C07176=1030.906,187.234,-109.081,169.495,44.538,158.415
C07177=1030.900,186.985,-109.057,169.491,44.540,158.415
C07178=1030.894,186.736,-109.033,169.489,44.542,158.415
C07179=1030.888,186.488,-109.009,169.485,44.543,158.415
C07180=1030.882,186.238,-108.984,169.482,44.545,158.415
C07181=1030.877,185.990,-108.961,169.478,44.546,158.415
C07182=1030.870,185.741,-108.938,169.475,44.549,158.415
C07183=1030.865,185.492,-108.913,169.472,44.550,158.415
C07184=1030.859,185.244,-108.889,169.468,44.552,158.415
C07185=1030.854,184.995,-108.866,169.466,44.553,158.415
C07186=1030.847,184.746,-108.842,169.462,44.555,158.415
C07187=1030.842,184.497,-108.818,169.458,44.557,158.415
C07188=1030.836,184.249,-108.794,169.456,44.559,158.415
C07189=1030.829,183.999,-108.771,169.452,44.560,158.415
C07190=1030.824,183.751,-108.746,169.449,44.562,158.415
C07191=1030.818,183.502,-108.723,169.445,44.564,158.415
C07192=1030.813,183.253,-108.699,169.442,44.566,158.415
C07193=1030.806,183.004,-108.675,169.439,44.567,158.415
C07194=1030.800,182.756,-108.651,169.435,44.569,158.415
C07195=1030.795,182.507,-108.629,169.433,44.571,158.416
C07196=1030.788,182.257,-108.605,169.429,44.573,158.416
C07197=1030.781,182.009,-108.582,169.426,44.575,158.416
C07198=1030.776,181.760,-108.559,169.423,44.577,158.416
C07199=1030.769,181.511,-108.535,169.419,44.579,158.416
C07200=1030.763,181.263,-108.512,169.416,44.581,158.416
C07201=1030.758,181.014,-108.489,169.413,44.583,158.416
C07202=1030.751,180.765,-108.465,169.410,44.585,158.416
C07203=1030.744,180.516,-108.443,169.406,44.587,158.416
C07204=1030.739,180.267,-108.420,169.403,44.588,158.416
C07205=1030.732,180.018,-108.396,169.400,44.591,158.416
C07206=1030.726,179.769,-108.373,169.396,44.593,158.417
C07207=1030.720,179.521,-108.349,169.394,44.595,158.417
C07208=1030.714,179.271,-108.326,169.390,44.597,158.417
C07209=1030.708,179.023,-108.304,169.387,44.599,158.417
C07210=1030.702,178.774,-108.281,169.384,44.601,158.417
C07211=1030.696,178.526,-108.257,169.380,44.602,158.417
C07212=1030.689,178.276,-108.234,169.377,44.604,158.417
C07213=1030.684,178.027,-108.211,169.374,44.606,158.417
C07214=1030.677,177.779,-108.188,169.370,44.608,158.417
C07215=1030.671,177.530,-108.165,169.368,44.610,158.417
C07216=1030.665,177.281,-108.141,169.364,44.613,158.417
C07217=1030.659,177.032,-108.119,169.362,44.614,158.418
C07218=1030.653,176.783,-108.096,169.358,44.616,158.418
C07219=1030.647,176.535,-108.073,169.355,44.618,158.418
C07220=1030.640,176.285,-108.049,169.352,44.620,158.418
C07221=1030.635,176.036,-108.026,169.348,44.622,158.418
C07222=1030.629,175.788,-108.003,169.346,44.624,158.418
C07223=1030.623,175.539,-107.980,169.342,44.626,158.418
C07224=1030.616,175.291,-107.957,169.339,44.628,158.418
C07225=1030.610,175.041,-107.934,169.336,44.630,158.418
C07226=1030.604,174.792,-107.911,169.333,44.632,158.418
C07227=1030.599,174.543,-107.888,169.329,44.634,158.418
C07228=1030.593,174.294,-107.865,169.326,44.636,158.419
C07229=1030.586,174.046,-107.843,169.323,44.638,158.419
C07230=1030.581,173.797,-107.820,169.320,44.640,158.419
C07231=1030.574,173.548,-107.796,169.317,44.642,158.419
C07232=1030.568,173.299,-107.773,169.314,44.644,158.419
C07233=1030.563,173.050,-107.750,169.311,44.646,158.419
C07234=1030.556,172.766,-107.724,169.307,44.648,158.419
C07235=1030.549,172.483,-107.698,169.304,44.650,158.419
C07236=1030.542,172.199,-107.672,169.300,44.652,158.419
C07237=1030.535,171.914,-107.646,169.297,44.655,158.420
C07238=1030.529,171.665,-107.623,169.293,44.657,158.420
C07239=1030.524,171.417,-107.600,169.291,44.659,158.420
C07240=1030.517,171.168,-107.578,169.287,44.661,158.420
C07241=1030.511,170.919,-107.555,169.284,44.663,158.420
C07242=1030.506,170.670,-107.532,169.281,44.665,158.420
C07243=1030.499,170.421,-107.509,169.278,44.667,158.420
C07244=1030.494,170.172,-107.486,169.275,44.669,158.420
C07245=1030.487,169.923,-107.463,169.272,44.671,158.420
C07246=1030.481,169.674,-107.440,169.269,44.673,158.421
C07247=1030.476,169.425,-107.418,169.266,44.674,158.421
C07248=1030.470,169.176,-107.395,169.262,44.676,158.421
C07249=1030.463,168.928,-107.372,169.260,44.678,158.421
C07250=1030.458,168.679,-107.349,169.256,44.681,158.421
C07251=1030.452,168.430,-107.326,169.254,44.682,158.421
C07252=1030.446,168.181,-107.303,169.250,44.685,158.421
C07253=1030.440,167.933,-107.281,169.247,44.687,158.421
C07254=1030.434,167.683,-107.259,169.244,44.689,158.421
C07255=1030.429,167.434,-107.236,169.241,44.691,158.421
C07256=1030.423,167.185,-107.213,169.239,44.693,158.422
C07257=1030.416,166.937,-107.191,169.235,44.695,158.422
C07258=1030.411,166.688,-107.168,169.233,44.697,158.422
C07259=1030.405,166.439,-107.145,169.229,44.698,158.422
C07260=1030.399,166.190,-107.122,169.226,44.700,158.422
C07261=1030.393,165.941,-107.100,169.223,44.702,158.422
C07262=1030.387,165.692,-107.077,169.220,44.704,158.422
C07263=1030.382,165.443,-107.054,169.217,44.706,158.422
C07264=1030.376,165.194,-107.031,169.214,44.708,158.422
C07265=1030.369,164.945,-107.009,169.211,44.710,158.423
C07266=1030.364,164.696,-106.987,169.208,44.712,158.423
C07267=1030.358,164.447,-106.964,169.205,44.714,158.423
C07268=1030.353,164.199,-106.941,169.202,44.716,158.423
C07269=1030.347,163.950,-106.919,169.199,44.718,158.423
C07270=1030.341,163.701,-106.896,169.197,44.720,158.423
C07271=1030.335,163.452,-106.874,169.193,44.722,158.423
C07272=1030.330,163.203,-106.851,169.190,44.724,158.423
C07273=1030.323,162.954,-106.828,169.188,44.726,158.423
C07274=1030.318,162.705,-106.806,169.184,44.728,158.423
C07275=1030.312,162.456,-106.783,169.181,44.730,158.424
C07276=1030.306,162.207,-106.761,169.178,44.732,158.424
C07277=1030.300,161.958,-106.738,169.175,44.734,158.424
C07278=1030.295,161.710,-106.716,169.173,44.736,158.424
C07279=1030.289,161.461,-106.693,169.169,44.738,158.424
C07280=1030.283,161.212,-106.671,169.167,44.740,158.424
C07281=1030.277,160.963,-106.648,169.164,44.742,158.424
C07282=1030.272,160.714,-106.626,169.160,44.744,158.424
C07283=1030.266,160.465,-106.604,169.158,44.746,158.425
C07284=1030.260,160.216,-106.581,169.155,44.748,158.425
C07285=1030.255,159.967,-106.558,169.152,44.749,158.425
C07286=1030.249,159.718,-106.536,169.149,44.751,158.425
C07287=1030.243,159.469,-106.514,169.145,44.754,158.425
C07288=1030.237,159.220,-106.492,169.143,44.756,158.425
C07289=1030.231,158.971,-106.469,169.141,44.758,158.425
C07290=1030.225,158.722,-106.448,169.137,44.760,158.425
C07291=1030.218,158.473,-106.425,169.134,44.762,158.425
C07292=1030.213,158.224,-106.403,169.131,44.764,158.426
C07293=1030.207,157.975,-106.382,169.128,44.766,158.426
C07294=1030.201,157.727,-106.359,169.126,44.769,158.426
C07295=1030.195,157.477,-106.337,169.122,44.771,158.426
C07296=1030.189,157.229,-106.315,169.120,44.773,158.426
C07297=1030.183,156.980,-106.293,169.116,44.775,158.426
C07298=1030.176,156.695,-106.267,169.113,44.777,158.426
C07299=1030.170,156.411,-106.243,169.110,44.780,158.427
C07300=1030.162,156.127,-106.218,169.107,44.782,158.427
C07301=1030.156,155.842,-106.193,169.103,44.785,158.427
C07302=1030.149,155.593,-106.170,169.100,44.787,158.427
C07303=1030.144,155.344,-106.149,169.097,44.789,158.427
C07304=1030.138,155.095,-106.127,169.095,44.791,158.427
C07305=1030.132,154.846,-106.105,169.091,44.794,158.428
C07306=1030.126,154.597,-106.083,169.089,44.796,158.428
C07307=1030.120,154.348,-106.061,169.086,44.798,158.428
C07308=1030.115,154.099,-106.039,169.083,44.800,158.428
C07309=1030.108,153.851,-106.017,169.080,44.802,158.428
C07310=1030.102,153.601,-105.995,169.078,44.804,158.428
C07311=1030.096,153.352,-105.974,169.074,44.807,158.429
C07312=1030.091,153.103,-105.952,169.072,44.808,158.429
C07313=1030.085,152.855,-105.930,169.068,44.811,158.429
C07314=1030.078,152.606,-105.908,169.066,44.813,158.429
C07315=1030.072,152.356,-105.886,169.063,44.815,158.429
C07316=1030.066,152.107,-105.865,169.060,44.817,158.429
C07317=1030.060,151.859,-105.843,169.057,44.819,158.429
C07318=1030.054,151.609,-105.822,169.055,44.821,158.430
C07319=1030.049,151.360,-105.799,169.051,44.823,158.430
C07320=1030.042,151.111,-105.777,169.049,44.826,158.430
C07321=1030.037,150.863,-105.756,169.046,44.828,158.430
C07322=1030.031,150.614,-105.734,169.043,44.830,158.430
C07323=1030.025,150.364,-105.713,169.040,44.832,158.430
C07324=1030.018,150.115,-105.691,169.038,44.835,158.431
C07325=1030.013,149.867,-105.670,169.034,44.837,158.431
C07326=1030.007,149.617,-105.648,169.032,44.839,158.431
C07327=1030.000,149.368,-105.627,169.029,44.841,158.431
C07328=1029.996,149.119,-105.605,169.026,44.844,158.431
C07329=1029.989,148.870,-105.583,169.023,44.846,158.431
C07330=1029.983,148.621,-105.561,169.021,44.848,158.431
C07331=1029.977,148.373,-105.539,169.017,44.850,158.431
C07332=1029.971,148.124,-105.518,169.015,44.852,158.432
C07333=1029.965,147.875,-105.496,169.012,44.854,158.432
C07334=1029.959,147.626,-105.475,169.009,44.856,158.432
C07335=1029.953,147.377,-105.453,169.006,44.858,158.432
C07336=1029.948,147.127,-105.432,169.004,44.861,158.432
C07337=1029.941,146.878,-105.411,169.000,44.863,158.433
C07338=1029.936,146.629,-105.389,168.998,44.865,158.433
C07339=1029.930,146.380,-105.368,168.995,44.867,158.433
C07340=1029.924,146.131,-105.346,168.992,44.870,158.433
C07341=1029.918,145.883,-105.325,168.989,44.872,158.433
C07342=1029.912,145.633,-105.303,168.987,44.874,158.433
C07343=1029.905,145.384,-105.282,168.983,44.877,158.434
C07344=1029.899,145.136,-105.261,168.981,44.879,158.434
C07345=1029.893,144.887,-105.239,168.978,44.881,158.434
C07346=1029.887,144.637,-105.218,168.975,44.883,158.434
C07347=1029.882,144.388,-105.197,168.972,44.885,158.434
C07348=1029.876,144.139,-105.175,168.970,44.888,158.434
C07349=1029.869,143.890,-105.154,168.967,44.890,158.435
C07350=1029.863,143.642,-105.133,168.964,44.892,158.435
C07351=1029.857,143.392,-105.112,168.962,44.895,158.435
C07352=1029.852,143.143,-105.091,168.959,44.897,158.435
C07353=1029.846,142.894,-105.069,168.955,44.899,158.435
C07354=1029.839,142.645,-105.048,168.953,44.901,158.435
C07355=1029.834,142.397,-105.026,168.951,44.903,158.436
C07356=1029.828,142.147,-105.006,168.947,44.906,158.436
C07357=1029.822,141.899,-104.985,168.945,44.908,158.436
C07358=1029.815,141.649,-104.963,168.942,44.910,158.436
C07359=1029.809,141.400,-104.942,168.940,44.912,158.436
C07360=1029.804,141.151,-104.921,168.936,44.915,158.436
C07361=1029.798,140.902,-104.899,168.934,44.917,158.437
C07362=1029.791,140.618,-104.875,168.930,44.920,158.437
C07363=1029.784,140.333,-104.851,168.928,44.922,158.437
C07364=1029.778,140.047,-104.827,168.924,44.925,158.437
C07365=1029.771,139.763,-104.803,168.921,44.927,158.437
C07366=1029.765,139.514,-104.781,168.919,44.929,158.438
C07367=1029.759,139.265,-104.761,168.916,44.931,158.438
C07368=1029.753,139.016,-104.740,168.913,44.934,158.438
C07369=1029.747,138.768,-104.718,168.910,44.936,158.438
C07370=1029.741,138.518,-104.697,168.908,44.938,158.438
C07371=1029.735,138.269,-104.677,168.905,44.941,158.438
C07372=1029.729,138.020,-104.656,168.902,44.943,158.439
C07373=1029.723,137.770,-104.634,168.899,44.946,158.439
C07374=1029.717,137.522,-104.613,168.897,44.947,158.439
C07375=1029.711,137.272,-104.593,168.893,44.950,158.439
C07376=1029.705,137.024,-104.571,168.891,44.952,158.439
C07377=1029.699,136.774,-104.551,168.888,44.954,158.439
C07378=1029.693,136.526,-104.530,168.886,44.957,158.440
C07379=1029.687,136.276,-104.509,168.883,44.959,158.440
C07380=1029.681,136.028,-104.488,168.880,44.962,158.440
C07381=1029.675,135.778,-104.467,168.878,44.964,158.440
C07382=1029.669,135.530,-104.446,168.875,44.966,158.440
C07383=1029.663,135.280,-104.426,168.872,44.968,158.441
C07384=1029.657,135.032,-104.404,168.869,44.970,158.441
C07385=1029.651,134.782,-104.384,168.867,44.973,158.441
C07386=1029.645,134.534,-104.363,168.864,44.975,158.441
C07387=1029.638,134.284,-104.342,168.861,44.978,158.441
C07388=1029.633,134.035,-104.322,168.859,44.980,158.442
C07389=1029.627,133.786,-104.300,168.856,44.982,158.442
C07390=1029.621,133.537,-104.280,168.854,44.984,158.442
C07391=1029.615,133.288,-104.259,168.850,44.987,158.442
C07392=1029.609,133.039,-104.239,168.848,44.989,158.442
C07393=1029.603,132.789,-104.218,168.845,44.991,158.442
C07394=1029.597,132.541,-104.197,168.843,44.994,158.443
C07395=1029.591,132.292,-104.176,168.839,44.996,158.443
C07396=1029.585,132.043,-104.155,168.837,44.999,158.443
C07397=1029.579,131.794,-104.135,168.834,45.001,158.443
C07398=1029.573,131.544,-104.114,168.832,45.003,158.443
C07399=1029.567,131.296,-104.093,168.830,45.005,158.444
C07400=1029.561,131.046,-104.072,168.826,45.007,158.444
C07401=1029.555,130.797,-104.052,168.824,45.010,158.444
C07402=1029.550,130.549,-104.031,168.821,45.012,158.444
C07403=1029.543,130.299,-104.011,168.819,45.015,158.444
C07404=1029.538,130.050,-103.990,168.815,45.017,158.445
C07405=1029.531,129.800,-103.970,168.813,45.019,158.445
C07406=1029.525,129.552,-103.950,168.810,45.021,158.445
C07407=1029.518,129.303,-103.929,168.808,45.024,158.445
C07408=1029.513,129.054,-103.908,168.805,45.027,158.445
C07409=1029.507,128.804,-103.888,168.802,45.029,158.446
C07410=1029.501,128.555,-103.868,168.800,45.032,158.446
C07411=1029.494,128.306,-103.848,168.797,45.033,158.446
C07412=1029.488,128.057,-103.828,168.794,45.036,158.446
C07413=1029.482,127.808,-103.807,168.792,45.038,158.446
C07414=1029.476,127.559,-103.786,168.789,45.041,158.447
C07415=1029.470,127.310,-103.766,168.787,45.044,158.447
C07416=1029.463,127.061,-103.746,168.783,45.046,158.447
C07417=1029.458,126.811,-103.725,168.781,45.048,158.447
C07418=1029.452,126.563,-103.705,168.779,45.050,158.447
C07419=1029.445,126.313,-103.685,168.776,45.053,158.448
C07420=1029.439,126.064,-103.665,168.773,45.056,158.448
C07421=1029.434,125.814,-103.644,168.770,45.058,158.448
C07422=1029.427,125.566,-103.624,168.768,45.060,158.448
C07423=1029.421,125.317,-103.604,168.766,45.062,158.448
C07424=1029.415,125.068,-103.583,168.763,45.065,158.449
C07425=1029.409,124.819,-103.563,168.760,45.067,158.449
C07426=1029.403,124.575,-103.543,168.757,45.070,158.449
C07427=1029.397,124.332,-103.524,168.755,45.072,158.449
C07428=1029.391,124.088,-103.504,168.752,45.075,158.450
C07429=1029.386,123.845,-103.484,168.750,45.077,158.450
C07430=1029.380,123.602,-103.464,168.748,45.079,158.450
C07431=1029.374,123.358,-103.445,168.744,45.081,158.450
C07432=1029.368,123.115,-103.425,168.742,45.084,158.450
C07433=1029.362,122.871,-103.405,168.739,45.086,158.450
C07434=1029.356,122.622,-103.385,168.737,45.089,158.451
C07435=1029.350,122.373,-103.365,168.734,45.091,158.451
C07436=1029.344,122.124,-103.345,168.732,45.093,158.451
C07437=1029.337,121.875,-103.325,168.728,45.095,158.451
C07438=1029.332,121.625,-103.304,168.726,45.098,158.451
C07439=1029.326,121.377,-103.284,168.724,45.101,158.452
C07440=1029.320,121.127,-103.264,168.721,45.103,158.452
C07441=1029.314,120.878,-103.244,168.719,45.105,158.452
C07442=1029.308,120.629,-103.223,168.716,45.107,158.452
C07443=1029.302,120.380,-103.203,168.713,45.110,158.453
C07444=1029.296,120.131,-103.183,168.711,45.112,158.453
C07445=1029.290,119.882,-103.163,168.708,45.115,158.453
C07446=1029.284,119.633,-103.144,168.706,45.117,158.453
C07447=1029.279,119.383,-103.123,168.703,45.119,158.453
C07448=1029.272,119.134,-103.103,168.701,45.121,158.454
C07449=1029.266,118.885,-103.083,168.698,45.124,158.454
C07450=1029.260,118.636,-103.063,168.695,45.126,158.454
C07451=1029.254,118.388,-103.043,168.693,45.129,158.454
C07452=1029.248,118.138,-103.022,168.690,45.131,158.454
C07453=1029.242,117.889,-103.002,168.688,45.134,158.455
C07454=1029.235,117.592,-102.979,168.685,45.136,158.455
C07455=1029.229,117.296,-102.955,168.681,45.139,158.455
C07456=1029.221,117.001,-102.931,168.679,45.142,158.455
C07457=1029.214,116.704,-102.907,168.676,45.145,158.456
C07458=1029.208,116.455,-102.887,168.673,45.147,158.456
C07459=1029.202,116.206,-102.867,168.671,45.149,158.456
C07460=1029.197,115.957,-102.848,168.668,45.151,158.456
C07461=1029.190,115.707,-102.828,168.665,45.154,158.456
C07462=1029.185,115.458,-102.807,168.662,45.156,158.456
C07463=1029.179,115.209,-102.787,168.660,45.159,158.457
C07464=1029.173,114.960,-102.768,168.658,45.161,158.457
C07465=1029.167,114.711,-102.748,168.655,45.164,158.457
C07466=1029.161,114.462,-102.728,168.653,45.165,158.457
C07467=1029.155,114.213,-102.708,168.650,45.167,158.457
C07468=1029.150,113.963,-102.688,168.648,45.170,158.458
C07469=1029.144,113.714,-102.668,168.644,45.172,158.458
C07470=1029.138,113.465,-102.648,168.642,45.175,158.458
C07471=1029.132,113.217,-102.628,168.639,45.177,158.458
C07472=1029.126,112.967,-102.609,168.637,45.180,158.458
C07473=1029.119,112.718,-102.588,168.635,45.182,158.459
C07474=1029.114,112.468,-102.569,168.632,45.184,158.459
C07475=1029.108,112.219,-102.549,168.630,45.187,158.459
C07476=1029.102,111.971,-102.529,168.627,45.189,158.459
C07477=1029.096,111.721,-102.510,168.624,45.192,158.459
C07478=1029.090,111.472,-102.490,168.622,45.194,158.460
C07479=1029.084,111.222,-102.470,168.619,45.196,158.460
C07480=1029.078,110.973,-102.450,168.617,45.199,158.460
C07481=1029.072,110.724,-102.431,168.614,45.201,158.460
C07482=1029.065,110.475,-102.412,168.612,45.204,158.461
C07483=1029.059,110.227,-102.392,168.610,45.206,158.461
C07484=1029.054,109.977,-102.373,168.606,45.209,158.461
C07485=1029.048,109.728,-102.353,168.604,45.211,158.461
C07486=1029.041,109.478,-102.333,168.601,45.213,158.461
C07487=1029.035,109.229,-102.314,168.599,45.216,158.462
C07488=1029.029,108.980,-102.294,168.597,45.219,158.462
C07489=1029.023,108.731,-102.275,168.594,45.220,158.462
C07490=1029.016,108.447,-102.253,168.591,45.223,158.462
C07491=1029.009,108.162,-102.231,168.588,45.227,158.463
C07492=1029.002,107.877,-102.209,168.586,45.230,158.463
C07493=1028.995,107.591,-102.186,168.582,45.232,158.463
C07494=1028.989,107.342,-102.166,168.580,45.234,158.463
C07495=1028.983,107.093,-102.147,168.577,45.237,158.463
C07496=1028.977,106.844,-102.128,168.575,45.240,158.464
C07497=1028.971,106.595,-102.108,168.573,45.242,158.464
C07498=1028.965,106.345,-102.089,168.569,45.245,158.464
C07499=1028.959,106.096,-102.071,168.567,45.247,158.464
C07500=1028.953,105.847,-102.051,168.564,45.249,158.464
C07501=1028.947,105.598,-102.031,168.562,45.252,158.465
C07502=1028.941,105.349,-102.011,168.560,45.254,158.465
C07503=1028.935,105.100,-101.993,168.557,45.257,158.465
C07504=1028.929,104.851,-101.973,168.555,45.259,158.465
C07505=1028.922,104.601,-101.953,168.553,45.261,158.466
C07506=1028.916,104.352,-101.935,168.549,45.264,158.466
C07507=1028.910,104.102,-101.915,168.547,45.267,158.466
C07508=1028.905,103.853,-101.896,168.544,45.269,158.466
C07509=1028.899,103.604,-101.876,168.542,45.271,158.466
C07510=1028.892,103.355,-101.857,168.540,45.273,158.467
C07511=1028.886,103.106,-101.838,168.537,45.276,158.467
C07512=1028.880,102.857,-101.818,168.535,45.279,158.467
C07513=1028.874,102.608,-101.800,168.532,45.281,158.467
C07514=1028.868,102.358,-101.780,168.530,45.283,158.468
C07515=1028.863,102.109,-101.761,168.527,45.286,158.468
C07516=1028.857,101.860,-101.741,168.524,45.288,158.468
C07517=1028.850,101.611,-101.722,168.522,45.291,158.468
C07518=1028.845,101.362,-101.703,168.519,45.293,158.468
C07519=1028.839,101.112,-101.684,168.517,45.296,158.469
C07520=1028.832,100.864,-101.665,168.515,45.298,158.469
C07521=1028.826,100.614,-101.645,168.512,45.300,158.469
C07522=1028.821,100.365,-101.626,168.510,45.303,158.469
C07523=1028.815,100.115,-101.607,168.507,45.305,158.469
C07524=1028.809,99.866,-101.588,168.505,45.308,158.470
C07525=1028.803,99.617,-101.569,168.502,45.310,158.470
C07526=1028.796,99.368,-101.550,168.499,45.312,158.470
C07527=1028.791,99.119,-101.530,168.497,45.315,158.470
C07528=1028.784,98.870,-101.512,168.495,45.318,158.471
C07529=1028.778,98.621,-101.493,168.492,45.320,158.471
C07530=1028.772,98.371,-101.474,168.490,45.322,158.471
C07531=1028.766,98.122,-101.455,168.488,45.325,158.471
C07532=1028.760,97.873,-101.436,168.484,45.328,158.471
C07533=1028.753,97.623,-101.417,168.482,45.330,158.472
C07534=1028.748,97.374,-101.398,168.479,45.333,158.472
C07535=1028.741,97.125,-101.379,168.477,45.335,158.472
C07536=1028.735,96.876,-101.361,168.475,45.337,158.472
C07537=1028.729,96.626,-101.342,168.472,45.340,158.473
C07538=1028.723,96.378,-101.323,168.470,45.343,158.473
C07539=1028.718,96.128,-101.304,168.468,45.345,158.473
C07540=1028.711,95.879,-101.285,168.464,45.348,158.473
C07541=1028.705,95.630,-101.267,168.462,45.350,158.473
C07542=1028.699,95.381,-101.247,168.460,45.353,158.474
C07543=1028.693,95.132,-101.229,168.457,45.355,158.474
C07544=1028.687,94.882,-101.210,168.455,45.358,158.474
C07545=1028.681,94.633,-101.191,168.452,45.360,158.474
C07546=1028.675,94.384,-101.172,168.450,45.362,158.474
C07547=1028.669,94.135,-101.153,168.448,45.365,158.475
C07548=1028.662,93.885,-101.134,168.445,45.368,158.475
C07549=1028.656,93.636,-101.115,168.443,45.370,158.475
C07550=1028.651,93.388,-101.097,168.439,45.373,158.475
C07551=1028.645,93.138,-101.078,168.437,45.375,158.476
C07552=1028.638,92.889,-101.059,168.435,45.377,158.476
C07553=1028.632,92.639,-101.041,168.432,45.380,158.476
C07554=1028.626,92.354,-101.019,168.430,45.383,158.476
C07555=1028.619,92.069,-100.997,168.427,45.385,158.477
C07556=1028.611,91.784,-100.976,168.424,45.388,158.477
C07557=1028.605,91.500,-100.955,168.421,45.391,158.477
C07558=1028.599,91.251,-100.936,168.419,45.394,158.477
C07559=1028.593,91.001,-100.917,168.416,45.396,158.477
C07560=1028.587,90.752,-100.898,168.414,45.398,158.478
C07561=1028.581,90.502,-100.880,168.412,45.401,158.478
C07562=1028.575,90.253,-100.861,168.409,45.403,158.478
C07563=1028.568,90.004,-100.842,168.407,45.406,158.478
C07564=1028.563,89.755,-100.824,168.405,45.408,158.479
C07565=1028.557,89.506,-100.805,168.401,45.411,158.479
C07566=1028.551,89.256,-100.787,168.399,45.413,158.479
C07567=1028.544,89.007,-100.768,168.397,45.416,158.479
C07568=1028.538,88.758,-100.750,168.394,45.419,158.480
C07569=1028.533,88.508,-100.731,168.392,45.421,158.480
C07570=1028.526,88.259,-100.712,168.389,45.423,158.480
C07571=1028.520,88.010,-100.694,168.387,45.426,158.480
C07572=1028.514,87.761,-100.676,168.385,45.429,158.480
C07573=1028.508,87.511,-100.658,168.381,45.431,158.481
C07574=1028.501,87.262,-100.639,168.379,45.434,158.481
C07575=1028.495,87.013,-100.621,168.377,45.436,158.481
C07576=1028.489,86.763,-100.602,168.374,45.439,158.481
C07577=1028.483,86.515,-100.584,168.372,45.442,158.482
C07578=1028.478,86.265,-100.566,168.370,45.444,158.482
C07579=1028.471,86.016,-100.547,168.367,45.446,158.482
C07580=1028.465,85.767,-100.528,168.365,45.449,158.482
C07581=1028.459,85.517,-100.510,168.363,45.452,158.483
C07582=1028.453,85.269,-100.492,168.359,45.454,158.483
C07583=1028.446,85.019,-100.473,168.357,45.457,158.483
C07584=1028.440,84.770,-100.455,168.355,45.459,158.483
C07585=1028.434,84.521,-100.437,168.352,45.461,158.483
C07586=1028.428,84.271,-100.419,168.350,45.464,158.484
C07587=1028.422,84.022,-100.401,168.347,45.467,158.484
C07588=1028.416,83.773,-100.383,168.345,45.469,158.484
C07589=1028.410,83.523,-100.363,168.343,45.471,158.484
C07590=1028.404,83.274,-100.345,168.340,45.474,158.484
C07591=1028.398,83.025,-100.327,168.338,45.477,158.485
C07592=1028.392,82.776,-100.309,168.335,45.479,158.485
C07593=1028.386,82.526,-100.291,168.332,45.482,158.485
C07594=1028.379,82.277,-100.272,168.330,45.484,158.485
C07595=1028.374,82.028,-100.254,168.328,45.487,158.486
C07596=1028.367,81.779,-100.236,168.325,45.489,158.486
C07597=1028.361,81.529,-100.218,168.323,45.492,158.486
C07598=1028.355,81.280,-100.199,168.321,45.494,158.486
C07599=1028.349,81.031,-100.182,168.318,45.496,158.486
C07600=1028.343,80.782,-100.163,168.316,45.499,158.487
C07601=1028.337,80.532,-100.144,168.313,45.502,158.487
C07602=1028.331,80.283,-100.126,168.311,45.504,158.487
C07603=1028.325,80.034,-100.108,168.309,45.506,158.487
C07604=1028.319,79.785,-100.090,168.306,45.509,158.488
C07605=1028.313,79.535,-100.072,168.303,45.511,158.488
C07606=1028.307,79.286,-100.053,168.301,45.514,158.488
C07607=1028.301,79.037,-100.035,168.298,45.517,158.488
C07608=1028.295,78.787,-100.018,168.296,45.519,158.488
C07609=1028.289,78.539,-99.999,168.293,45.521,158.489
C07610=1028.283,78.289,-99.981,168.291,45.524,158.489
C07611=1028.276,78.040,-99.963,168.289,45.526,158.489
C07612=1028.271,77.791,-99.945,168.286,45.529,158.489
C07613=1028.265,77.541,-99.927,168.284,45.532,158.490
C07614=1028.258,77.292,-99.909,168.281,45.534,158.490
C07615=1028.253,77.043,-99.891,168.279,45.536,158.490
C07616=1028.247,76.793,-99.873,168.277,45.539,158.490
C07617=1028.240,76.544,-99.854,168.275,45.542,158.490
C07618=1028.234,76.259,-99.834,168.271,45.545,158.491
C07619=1028.226,75.974,-99.813,168.268,45.547,158.491
C07620=1028.219,75.689,-99.793,168.266,45.550,158.491
C07621=1028.213,75.403,-99.773,168.262,45.553,158.491
C07622=1028.206,75.154,-99.754,168.260,45.556,158.492
C07623=1028.199,74.905,-99.737,168.258,45.558,158.492
C07624=1028.194,74.656,-99.720,168.256,45.561,158.492
C07625=1028.188,74.406,-99.702,168.253,45.563,158.492
C07626=1028.182,74.158,-99.683,168.251,45.566,158.493
C07627=1028.176,73.908,-99.665,168.249,45.569,158.493
C07628=1028.169,73.659,-99.648,168.246,45.571,158.493
C07629=1028.163,73.409,-99.631,168.244,45.573,158.493
C07630=1028.157,73.160,-99.613,168.240,45.576,158.493
C07631=1028.151,72.911,-99.594,168.238,45.579,158.494
C07632=1028.145,72.662,-99.576,168.236,45.581,158.494
C07633=1028.139,72.412,-99.559,168.233,45.584,158.494
C07634=1028.133,72.163,-99.541,168.231,45.586,158.494
C07635=1028.127,71.913,-99.524,168.229,45.589,158.495
C07636=1028.120,71.664,-99.505,168.226,45.591,158.495
C07637=1028.115,71.415,-99.487,168.224,45.594,158.495
C07638=1028.108,71.166,-99.470,168.222,45.596,158.495
C07639=1028.103,70.917,-99.452,168.219,45.599,158.496
C07640=1028.096,70.667,-99.434,168.217,45.601,158.496
C07641=1028.090,70.418,-99.417,168.215,45.604,158.496
C07642=1028.084,70.169,-99.400,168.211,45.607,158.496
C07643=1028.078,69.919,-99.382,168.209,45.609,158.496
C07644=1028.072,69.670,-99.364,168.206,45.611,158.496
C07645=1028.065,69.421,-99.346,168.204,45.614,158.497
C07646=1028.060,69.172,-99.328,168.202,45.617,158.497
C07647=1028.054,68.922,-99.311,168.199,45.619,158.497
C07648=1028.047,68.672,-99.293,168.197,45.622,158.497
C07649=1028.041,68.424,-99.276,168.195,45.624,158.498
C07650=1028.035,68.174,-99.258,168.193,45.627,158.498
C07651=1028.029,67.925,-99.241,168.190,45.629,158.498
C07652=1028.023,67.675,-99.223,168.188,45.632,158.498
C07653=1028.017,67.426,-99.205,168.184,45.635,158.499
C07654=1028.010,67.177,-99.188,168.182,45.637,158.499
C07655=1028.005,66.928,-99.170,168.180,45.639,158.499
C07656=1027.999,66.678,-99.152,168.177,45.642,158.499
C07657=1027.992,66.429,-99.135,168.175,45.645,158.499
C07658=1027.986,66.180,-99.117,168.173,45.647,158.500
C07659=1027.979,65.930,-99.100,168.170,45.649,158.500
C07660=1027.974,65.681,-99.083,168.168,45.652,158.500
C07661=1027.967,65.431,-99.066,168.166,45.655,158.500
C07662=1027.962,65.182,-99.048,168.163,45.658,158.501
C07663=1027.955,64.933,-99.031,168.160,45.660,158.501
C07664=1027.950,64.684,-99.013,168.158,45.663,158.501
C07665=1027.943,64.434,-98.996,168.155,45.665,158.501
C07666=1027.937,64.185,-98.979,168.153,45.668,158.501
C07667=1027.931,63.935,-98.961,168.150,45.670,158.502
C07668=1027.925,63.687,-98.944,168.148,45.673,158.502
C07669=1027.919,63.437,-98.926,168.146,45.675,158.502
C07670=1027.913,63.188,-98.909,168.144,45.678,158.502
C07671=1027.906,62.938,-98.892,168.141,45.681,158.503
C07672=1027.900,62.689,-98.875,168.138,45.684,158.503
C07673=1027.893,62.440,-98.857,168.136,45.686,158.503
C07674=1027.887,62.190,-98.841,168.133,45.688,158.503
C07675=1027.881,61.941,-98.824,168.131,45.691,158.504
C07676=1027.875,61.692,-98.806,168.129,45.694,158.504
C07677=1027.869,61.442,-98.789,168.126,45.697,158.504
C07678=1027.862,61.193,-98.772,168.124,45.699,158.504
C07679=1027.856,60.943,-98.755,168.121,45.702,158.505
C07680=1027.850,60.695,-98.738,168.119,45.705,158.505
C07681=1027.843,60.445,-98.721,168.116,45.708,158.505
C07682=1027.836,60.160,-98.702,168.113,45.711,158.505
C07683=1027.829,59.874,-98.681,168.111,45.713,158.506
C07684=1027.822,59.590,-98.662,168.107,45.716,158.506
C07685=1027.816,59.304,-98.643,168.105,45.720,158.506
C07686=1027.809,59.055,-98.625,168.103,45.722,158.506
C07687=1027.803,58.806,-98.609,168.100,45.725,158.506
C07688=1027.796,58.556,-98.592,168.097,45.727,158.507
C07689=1027.790,58.307,-98.574,168.095,45.730,158.507
C07690=1027.784,58.057,-98.558,168.093,45.733,158.507
C07691=1027.778,57.808,-98.541,168.091,45.735,158.508
C07692=1027.772,57.559,-98.524,168.088,45.738,158.508
C07693=1027.765,57.309,-98.506,168.086,45.740,158.508
C07694=1027.759,57.060,-98.489,168.082,45.743,158.508
C07695=1027.753,56.810,-98.473,168.080,45.746,158.508
C07696=1027.746,56.562,-98.456,168.078,45.748,158.509
C07697=1027.740,56.312,-98.439,168.076,45.751,158.509
C07698=1027.734,56.063,-98.422,168.073,45.754,158.509
C07699=1027.728,55.814,-98.405,168.071,45.756,158.509
C07700=1027.722,55.564,-98.388,168.069,45.759,158.510
C07701=1027.715,55.315,-98.371,168.066,45.761,158.510
C07702=1027.710,55.065,-98.354,168.063,45.764,158.510
C07703=1027.703,54.816,-98.337,168.061,45.767,158.510
C07704=1027.697,54.567,-98.321,168.058,45.769,158.510
C07705=1027.690,54.317,-98.303,168.056,45.772,158.511
C07706=1027.685,54.068,-98.286,168.054,45.774,158.511
C07707=1027.679,53.819,-98.270,168.051,45.777,158.511
C07708=1027.672,53.569,-98.253,168.049,45.780,158.511
C07709=1027.666,53.320,-98.236,168.047,45.782,158.512
C07710=1027.661,53.070,-98.219,168.043,45.785,158.512
C07711=1027.654,52.821,-98.202,168.041,45.788,158.512
C07712=1027.648,52.572,-98.185,168.039,45.790,158.512
C07713=1027.642,52.323,-98.168,168.036,45.792,158.512
C07714=1027.635,52.073,-98.152,168.034,45.795,158.513
C07715=1027.630,51.824,-98.134,168.032,45.798,158.513
C07716=1027.624,51.574,-98.118,168.029,45.801,158.513
C07717=1027.617,51.325,-98.101,168.027,45.803,158.513
C07718=1027.611,51.076,-98.084,168.025,45.805,158.514
C07719=1027.605,50.827,-98.067,168.021,45.808,158.514
C07720=1027.599,50.577,-98.050,168.019,45.811,158.514
C07721=1027.593,50.327,-98.034,168.016,45.813,158.514
C07722=1027.587,50.079,-98.017,168.014,45.816,158.514
C07723=1027.581,49.829,-98.001,168.012,45.818,158.515
C07724=1027.575,49.579,-97.983,168.009,45.820,158.515
C07725=1027.569,49.330,-97.967,168.007,45.823,158.515
C07726=1027.563,49.081,-97.950,168.005,45.826,158.515
C07727=1027.556,48.832,-97.933,168.003,45.829,158.516
C07728=1027.550,48.582,-97.917,168.000,45.831,158.516
C07729=1027.544,48.333,-97.899,167.997,45.834,158.516
C07730=1027.538,48.084,-97.883,167.994,45.836,158.516
C07731=1027.532,47.834,-97.866,167.992,45.838,158.516
C07732=1027.526,47.585,-97.849,167.990,45.841,158.516
C07733=1027.520,47.335,-97.833,167.987,45.844,158.517
C07734=1027.514,47.086,-97.816,167.985,45.846,158.517
C07735=1027.508,46.837,-97.799,167.983,45.849,158.517
C07736=1027.502,46.587,-97.783,167.980,45.851,158.517
C07737=1027.496,46.338,-97.766,167.978,45.853,158.517
C07738=1027.489,46.089,-97.749,167.976,45.856,158.518
C07739=1027.484,45.839,-97.733,167.973,45.859,158.518
C07740=1027.478,45.589,-97.716,167.971,45.861,158.518
C07741=1027.472,45.340,-97.700,167.967,45.864,158.518
C07742=1027.466,45.091,-97.683,167.965,45.866,158.519
C07743=1027.460,44.842,-97.666,167.963,45.869,158.519
C07744=1027.454,44.592,-97.650,167.960,45.871,158.519
C07745=1027.448,44.343,-97.633,167.958,45.873,158.519
C07746=1027.441,44.057,-97.614,167.956,45.876,158.519
C07747=1027.434,43.772,-97.594,167.952,45.879,158.519
C07748=1027.428,43.486,-97.576,167.950,45.882,158.520
C07749=1027.420,43.201,-97.557,167.947,45.885,158.520
C07750=1027.415,42.951,-97.540,167.944,45.887,158.520
C07751=1027.409,42.702,-97.524,167.942,45.890,158.520
C07752=1027.403,42.452,-97.507,167.940,45.893,158.521
C07753=1027.396,42.203,-97.492,167.937,45.895,158.521
C07754=1027.389,41.953,-97.475,167.934,45.898,158.521
C07755=1027.383,41.705,-97.458,167.932,45.901,158.521
C07756=1027.377,41.455,-97.442,167.930,45.903,158.522
C07757=1027.371,41.206,-97.426,167.927,45.905,158.522
C07758=1027.365,40.957,-97.409,167.925,45.908,158.522
C07759=1027.359,40.707,-97.393,167.923,45.911,158.522
C07760=1027.353,40.457,-97.376,167.920,45.914,158.522
C07761=1027.347,40.208,-97.360,167.918,45.916,158.523
C07762=1027.341,39.958,-97.344,167.914,45.919,158.523
C07763=1027.335,39.709,-97.328,167.912,45.921,158.523
C07764=1027.328,39.460,-97.312,167.910,45.924,158.523
C07765=1027.322,39.211,-97.296,167.907,45.926,158.523
C07766=1027.316,38.961,-97.280,167.905,45.929,158.524
C07767=1027.310,38.711,-97.263,167.903,45.931,158.524
C07768=1027.304,38.462,-97.247,167.901,45.934,158.524
C07769=1027.298,38.213,-97.230,167.898,45.936,158.524
C07770=1027.292,37.963,-97.214,167.895,45.939,158.524
C07771=1027.286,37.714,-97.198,167.893,45.942,158.525
C07772=1027.280,37.465,-97.182,167.890,45.944,158.525
C07773=1027.274,37.215,-97.165,167.888,45.947,158.525
C07774=1027.268,36.966,-97.149,167.885,45.949,158.525
C07775=1027.261,36.716,-97.133,167.883,45.952,158.526
C07776=1027.255,36.467,-97.117,167.881,45.954,158.526
C07777=1027.249,36.217,-97.101,167.877,45.957,158.526
C07778=1027.242,35.968,-97.085,167.875,45.960,158.526
C07779=1027.237,35.718,-97.069,167.873,45.963,158.526
C07780=1027.231,35.469,-97.053,167.871,45.965,158.527
C07781=1027.224,35.220,-97.037,167.868,45.968,158.527
C07782=1027.218,34.971,-97.021,167.865,45.970,158.527
C07783=1027.212,34.721,-97.005,167.862,45.973,158.527
C07784=1027.205,34.472,-96.989,167.860,45.976,158.527
C07785=1027.200,34.222,-96.974,167.858,45.979,158.528
C07786=1027.193,33.972,-96.957,167.856,45.981,158.528
C07787=1027.187,33.723,-96.941,167.853,45.983,158.528
C07788=1027.181,33.474,-96.925,167.850,45.986,158.528
C07789=1027.175,33.225,-96.909,167.848,45.989,158.528
C07790=1027.168,32.975,-96.894,167.845,45.992,158.529
C07791=1027.162,32.726,-96.878,167.843,45.995,158.529
C07792=1027.156,32.476,-96.861,167.841,45.997,158.529
C07793=1027.150,32.227,-96.846,167.838,45.999,158.529
C07794=1027.144,31.978,-96.830,167.835,46.002,158.530
C07795=1027.138,31.728,-96.814,167.833,46.005,158.530
C07796=1027.131,31.479,-96.798,167.830,46.007,158.530
C07797=1027.125,31.230,-96.782,167.828,46.010,158.530
C07798=1027.119,30.980,-96.766,167.826,46.013,158.530
C07799=1027.113,30.730,-96.751,167.823,46.015,158.531
C07800=1027.107,30.481,-96.735,167.820,46.018,158.531
C07801=1027.100,30.232,-96.719,167.818,46.020,158.531
C07802=1027.095,29.982,-96.703,167.815,46.023,158.531
C07803=1027.089,29.733,-96.687,167.813,46.026,158.531
C07804=1027.082,29.484,-96.672,167.811,46.028,158.532
C07805=1027.077,29.234,-96.656,167.808,46.031,158.532
C07806=1027.071,28.984,-96.640,167.805,46.034,158.532
C07807=1027.064,28.735,-96.624,167.803,46.036,158.532
C07808=1027.058,28.485,-96.609,167.800,46.038,158.532
C07809=1027.052,28.236,-96.592,167.798,46.041,158.533
C07810=1027.045,27.951,-96.575,167.795,46.044,158.533
C07811=1027.038,27.665,-96.556,167.792,46.047,158.533
C07812=1027.031,27.380,-96.538,167.789,46.050,158.533
C07813=1027.024,27.094,-96.521,167.786,46.054,158.534
C07814=1027.018,26.845,-96.505,167.784,46.056,158.534
C07815=1027.011,26.596,-96.489,167.781,46.058,158.534
C07816=1027.005,26.346,-96.474,167.779,46.061,158.534
C07817=1026.999,26.097,-96.458,167.777,46.064,158.534
C07818=1026.993,25.847,-96.443,167.774,46.067,158.535
C07819=1026.987,25.598,-96.427,167.771,46.069,158.535
C07820=1026.980,25.348,-96.412,167.769,46.072,158.535
C07821=1026.974,25.099,-96.396,167.767,46.074,158.535
C07822=1026.968,24.849,-96.381,167.764,46.077,158.536
C07823=1026.961,24.600,-96.365,167.761,46.080,158.536
C07824=1026.956,24.350,-96.349,167.759,46.083,158.536
C07825=1026.949,24.101,-96.334,167.756,46.085,158.536
C07826=1026.944,23.852,-96.319,167.754,46.088,158.536
C07827=1026.937,23.602,-96.304,167.752,46.090,158.537
C07828=1026.932,23.353,-96.287,167.748,46.093,158.537
C07829=1026.925,23.103,-96.272,167.746,46.096,158.537
C07830=1026.918,22.854,-96.257,167.744,46.098,158.537
C07831=1026.913,22.604,-96.241,167.741,46.101,158.537
C07832=1026.906,22.355,-96.226,167.739,46.104,158.538
C07833=1026.900,22.105,-96.210,167.736,46.107,158.538
C07834=1026.894,21.855,-96.195,167.733,46.109,158.538
C07835=1026.888,21.607,-96.180,167.731,46.111,158.538
C07836=1026.882,21.357,-96.164,167.729,46.114,158.538
C07837=1026.876,21.108,-96.149,167.727,46.117,158.539
C07838=1026.869,20.858,-96.134,167.723,46.119,158.539
C07839=1026.864,20.608,-96.118,167.721,46.122,158.539
C07840=1026.857,20.359,-96.102,167.718,46.125,158.539
C07841=1026.851,20.109,-96.087,167.716,46.128,158.539
C07842=1026.845,19.860,-96.072,167.714,46.130,158.540
C07843=1026.839,19.611,-96.057,167.710,46.133,158.540
C07844=1026.833,19.361,-96.041,167.708,46.135,158.540
C07845=1026.827,19.112,-96.026,167.706,46.138,158.540
C07846=1026.820,18.863,-96.010,167.703,46.140,158.540
C07847=1026.814,18.613,-95.995,167.700,46.143,158.541
C07848=1026.808,18.363,-95.980,167.698,46.146,158.541
C07849=1026.802,18.114,-95.965,167.696,46.149,158.541
C07850=1026.796,17.865,-95.950,167.693,46.151,158.541
C07851=1026.790,17.615,-95.934,167.691,46.153,158.541
C07852=1026.784,17.365,-95.919,167.688,46.156,158.542
C07853=1026.777,17.116,-95.904,167.685,46.159,158.542
C07854=1026.771,16.866,-95.889,167.683,46.162,158.542
C07855=1026.765,16.618,-95.874,167.681,46.165,158.542
C07856=1026.759,16.368,-95.859,167.677,46.167,158.542
C07857=1026.753,16.118,-95.844,167.675,46.170,158.543
C07858=1026.746,15.868,-95.829,167.673,46.172,158.543
C07859=1026.740,15.619,-95.814,167.670,46.175,158.543
C07860=1026.735,15.370,-95.798,167.668,46.177,158.543
C07861=1026.728,15.121,-95.783,167.665,46.180,158.543
C07862=1026.722,14.871,-95.768,167.662,46.183,158.544
C07863=1026.715,14.621,-95.753,167.660,46.186,158.544
C07864=1026.710,14.372,-95.738,167.658,46.188,158.544
C07865=1026.704,14.122,-95.723,167.654,46.191,158.544
C07866=1026.698,13.873,-95.708,167.652,46.194,158.544
C07867=1026.691,13.624,-95.692,167.650,46.196,158.545
C07868=1026.685,13.375,-95.678,167.648,46.199,158.545
C07869=1026.679,13.125,-95.663,167.644,46.201,158.545
C07870=1026.672,12.875,-95.648,167.642,46.204,158.545
C07871=1026.666,12.626,-95.633,167.640,46.207,158.545
C07872=1026.660,12.376,-95.618,167.636,46.210,158.546
C07873=1026.654,12.127,-95.603,167.634,46.213,158.546
C07874=1026.647,11.843,-95.586,167.631,46.216,158.546
C07875=1026.639,11.558,-95.569,167.629,46.219,158.546
C07876=1026.633,11.274,-95.553,167.625,46.222,158.547
C07877=1026.626,10.990,-95.536,167.622,46.225,158.547
C07878=1026.619,10.740,-95.521,167.620,46.228,158.547
C07879=1026.613,10.490,-95.506,167.618,46.231,158.547
C07880=1026.607,10.241,-95.492,167.614,46.234,158.548
C07881=1026.601,9.992,-95.477,167.612,46.236,158.548
C07882=1026.594,9.742,-95.462,167.610,46.238,158.548
C07883=1026.588,9.493,-95.447,167.606,46.241,158.548
C07884=1026.582,9.244,-95.432,167.604,46.244,158.548
C07885=1026.576,8.994,-95.417,167.602,46.247,158.549
C07886=1026.569,8.744,-95.403,167.600,46.250,158.549
C07887=1026.563,8.495,-95.388,167.596,46.253,158.549
C07888=1026.557,8.246,-95.373,167.594,46.255,158.549
C07889=1026.550,7.996,-95.359,167.592,46.258,158.549
C07890=1026.545,7.747,-95.345,167.588,46.261,158.549
C07891=1026.538,7.497,-95.330,167.586,46.263,158.550
C07892=1026.532,7.247,-95.315,167.584,46.266,158.550
C07893=1026.526,6.998,-95.300,167.582,46.269,158.550
C07894=1026.520,6.749,-95.285,167.578,46.271,158.550
C07895=1026.513,6.498,-95.271,167.576,46.274,158.551
C07896=1026.508,6.250,-95.257,167.573,46.277,158.551
C07897=1026.501,6.000,-95.242,167.570,46.280,158.551
C07898=1026.496,5.751,-95.227,167.568,46.283,158.551
C07899=1026.489,5.501,-95.212,167.565,46.285,158.551
C07900=1026.483,5.252,-95.197,167.563,46.287,158.552
C07901=1026.477,5.002,-95.183,167.560,46.290,158.552
C07902=1026.471,4.752,-95.168,167.558,46.293,158.552
C07903=1026.465,4.503,-95.153,167.555,46.295,158.552
C07904=1026.459,4.254,-95.139,167.552,46.298,158.552
C07905=1026.452,4.004,-95.125,167.550,46.301,158.552
C07906=1026.446,3.755,-95.111,167.547,46.304,158.553
C07907=1026.440,3.505,-95.096,167.545,46.307,158.553
C07908=1026.434,3.256,-95.081,167.542,46.309,158.553
C07909=1026.428,3.006,-95.067,167.539,46.312,158.553
C07910=1026.422,2.756,-95.052,167.537,46.314,158.553
C07911=1026.416,2.507,-95.037,167.534,46.317,158.554
C07912=1026.409,2.258,-95.022,167.531,46.319,158.554
C07913=1026.404,2.008,-95.009,167.529,46.322,158.554
C07914=1026.398,1.758,-94.994,167.527,46.325,158.554
C07915=1026.392,1.510,-94.979,167.523,46.327,158.554
C07916=1026.386,1.259,-94.965,167.521,46.330,158.554
C07917=1026.379,1.010,-94.950,167.519,46.333,158.555
C07918=1026.373,0.761,-94.936,167.515,46.336,158.555
C07919=1026.367,0.511,-94.922,167.513,46.338,158.555
C07920=1026.361,0.262,-94.907,167.511,46.341,158.555
C07921=1026.355,0.012,-94.892,167.508,46.343,158.556
C07922=1026.349,-0.238,-94.878,167.505,46.346,158.556
C07923=1026.343,-0.487,-94.863,167.503,46.349,158.556
C07924=1026.337,-0.736,-94.849,167.500,46.351,158.556
C07925=1026.331,-0.986,-94.834,167.497,46.354,158.556
C07926=1026.325,-1.235,-94.820,167.495,46.356,158.556
C07927=1026.319,-1.486,-94.806,167.492,46.359,158.557
C07928=1026.312,-1.734,-94.792,167.490,46.362,158.557
C07929=1026.306,-1.984,-94.777,167.487,46.364,158.557
C07930=1026.301,-2.234,-94.763,167.484,46.367,158.557
C07931=1026.294,-2.483,-94.748,167.482,46.370,158.557
C07932=1026.289,-2.733,-94.734,167.480,46.372,158.557
C07933=1026.283,-2.982,-94.719,167.476,46.375,158.558
C07934=1026.277,-3.232,-94.705,167.474,46.378,158.558
C07935=1026.271,-3.481,-94.691,167.471,46.380,158.558
C07936=1026.265,-3.731,-94.676,167.468,46.383,158.558
C07937=1026.259,-3.980,-94.662,167.466,46.386,158.558
C07938=1026.252,-4.263,-94.646,167.463,46.389,158.558
C07939=1026.244,-4.544,-94.630,167.460,46.391,158.559
C07940=1026.238,-4.827,-94.614,167.457,46.394,158.559
C07941=1026.231,-5.110,-94.599,167.454,46.398,158.559
C07942=1026.224,-5.359,-94.584,167.452,46.400,158.559
C07943=1026.218,-5.609,-94.571,167.448,46.403,158.559
C07944=1026.212,-5.859,-94.557,167.446,46.406,158.560
C07945=1026.206,-6.108,-94.543,167.443,46.409,158.560
C07946=1026.199,-6.358,-94.528,167.441,46.412,158.560
C07947=1026.194,-6.607,-94.514,167.438,46.415,158.560
C07948=1026.187,-6.857,-94.500,167.435,46.418,158.561
C07949=1026.181,-7.106,-94.486,167.433,46.420,158.561
C07950=1026.175,-7.356,-94.473,167.430,46.422,158.561
C07951=1026.169,-7.605,-94.458,167.427,46.425,158.561
C07952=1026.163,-7.854,-94.445,167.425,46.428,158.561
C07953=1026.157,-8.105,-94.430,167.422,46.431,158.561
C07954=1026.150,-8.353,-94.417,167.419,46.434,158.562
C07955=1026.145,-8.603,-94.403,167.417,46.436,158.562
C07956=1026.138,-8.853,-94.389,167.414,46.439,158.562
C07957=1026.132,-9.103,-94.375,167.411,46.442,158.562
C07958=1026.125,-9.352,-94.361,167.409,46.445,158.562
C07959=1026.120,-9.601,-94.347,167.406,46.448,158.563
C07960=1026.114,-9.851,-94.333,167.403,46.450,158.563
C07961=1026.107,-10.101,-94.319,167.401,46.453,158.563
C07962=1026.102,-10.350,-94.305,167.398,46.456,158.563
C07963=1026.095,-10.599,-94.292,167.396,46.458,158.563
C07964=1026.089,-10.849,-94.277,167.392,46.461,158.563
C07965=1026.083,-11.099,-94.264,167.390,46.464,158.564
C07966=1026.078,-11.348,-94.250,167.387,46.466,158.564
C07967=1026.070,-11.598,-94.236,167.384,46.469,158.564
C07968=1026.065,-11.847,-94.222,167.382,46.472,158.564
C07969=1026.059,-12.096,-94.209,167.379,46.474,158.564
C07970=1026.053,-12.347,-94.194,167.376,46.477,158.565
C07971=1026.046,-12.596,-94.181,167.374,46.480,158.565
C07972=1026.041,-12.846,-94.167,167.372,46.483,158.565
C07973=1026.034,-13.095,-94.153,167.368,46.485,158.565
C07974=1026.028,-13.345,-94.139,167.366,46.488,158.565
C07975=1026.022,-13.594,-94.126,167.363,46.491,158.565
C07976=1026.016,-13.844,-94.112,167.360,46.494,158.566
C07977=1026.010,-14.093,-94.098,167.358,46.496,158.566
C07978=1026.004,-14.343,-94.085,167.355,46.499,158.566
C07979=1025.998,-14.592,-94.071,167.352,46.502,158.566
C07980=1025.992,-14.842,-94.057,167.350,46.504,158.566
C07981=1025.986,-15.091,-94.043,167.347,46.507,158.566
C07982=1025.980,-15.341,-94.029,167.344,46.510,158.567
C07983=1025.974,-15.590,-94.016,167.342,46.512,158.567
C07984=1025.968,-15.840,-94.002,167.339,46.515,158.567
C07985=1025.962,-16.089,-93.988,167.336,46.517,158.567
C07986=1025.955,-16.339,-93.975,167.333,46.521,158.567
C07987=1025.950,-16.590,-93.962,167.331,46.523,158.568
C07988=1025.943,-16.839,-93.948,167.328,46.526,158.568
C07989=1025.937,-17.088,-93.935,167.325,46.529,158.568
C07990=1025.931,-17.337,-93.922,167.322,46.532,158.568
C07991=1025.925,-17.588,-93.908,167.320,46.535,158.568
C07992=1025.919,-17.837,-93.894,167.318,46.538,158.569
C07993=1025.912,-18.086,-93.881,167.314,46.540,158.569
C07994=1025.906,-18.335,-93.868,167.312,46.543,158.569
C07995=1025.900,-18.586,-93.854,167.309,46.546,158.569
C07996=1025.894,-18.835,-93.840,167.306,46.549,158.569
C07997=1025.888,-19.084,-93.827,167.303,46.552,158.569
C07998=1025.882,-19.334,-93.814,167.301,46.555,158.570
C07999=1025.876,-19.584,-93.801,167.298,46.557,158.570
C08000=1025.870,-19.834,-93.787,167.295,46.560,158.570
C08001=1025.863,-20.083,-93.774,167.293,46.562,158.570
C08002=1025.856,-20.363,-93.759,167.289,46.565,158.570
C08003=1025.849,-20.644,-93.743,167.286,46.569,158.570
C08004=1025.843,-20.925,-93.729,167.283,46.572,158.571
C08005=1025.836,-21.205,-93.714,167.280,46.575,158.571
C08006=1025.829,-21.455,-93.700,167.278,46.578,158.571
C08007=1025.823,-21.705,-93.687,167.274,46.580,158.571
C08008=1025.818,-21.955,-93.674,167.272,46.583,158.571
C08009=1025.812,-22.204,-93.660,167.269,46.586,158.572
C08010=1025.806,-22.453,-93.647,167.266,46.589,158.572
C08011=1025.799,-22.702,-93.634,167.264,46.592,158.572
C08012=1025.794,-22.953,-93.621,167.261,46.594,158.572
C08013=1025.787,-23.203,-93.607,167.258,46.597,158.572
C08014=1025.781,-23.452,-93.594,167.255,46.600,158.572
C08015=1025.775,-23.701,-93.581,167.253,46.603,158.573
C08016=1025.769,-23.951,-93.568,167.250,46.606,158.573
C08017=1025.764,-24.201,-93.554,167.247,46.608,158.573
C08018=1025.757,-24.450,-93.541,167.245,46.611,158.573
C08019=1025.751,-24.699,-93.528,167.242,46.614,158.573
C08020=1025.745,-24.949,-93.515,167.239,46.617,158.574
C08021=1025.739,-25.198,-93.502,167.236,46.619,158.574
C08022=1025.734,-25.448,-93.488,167.234,46.622,158.574
C08023=1025.728,-25.698,-93.475,167.230,46.625,158.574
C08024=1025.721,-25.948,-93.462,167.228,46.628,158.574
C08025=1025.715,-26.197,-93.448,167.226,46.630,158.574
C08026=1025.710,-26.447,-93.435,167.222,46.633,158.574
C08027=1025.703,-26.696,-93.422,167.220,46.636,158.575
C08028=1025.697,-26.946,-93.409,167.217,46.639,158.575
C08029=1025.691,-27.196,-93.396,167.214,46.641,158.575
C08030=1025.685,-27.445,-93.383,167.211,46.644,158.575
C08031=1025.679,-27.695,-93.370,167.209,46.647,158.575
C08032=1025.673,-27.944,-93.357,167.206,46.650,158.576
C08033=1025.667,-28.194,-93.345,167.203,46.652,158.576
C08034=1025.661,-28.443,-93.331,167.200,46.655,158.576
C08035=1025.655,-28.693,-93.319,167.198,46.658,158.576
C08036=1025.649,-28.942,-93.305,167.195,46.661,158.576
C08037=1025.643,-29.192,-93.293,167.192,46.663,158.576
C08038=1025.636,-29.441,-93.280,167.189,46.666,158.577
C08039=1025.631,-29.691,-93.267,167.187,46.669,158.577
C08040=1025.624,-29.941,-93.254,167.183,46.672,158.577
C08041=1025.618,-30.190,-93.241,167.181,46.675,158.577
C08042=1025.612,-30.440,-93.228,167.178,46.678,158.577
C08043=1025.606,-30.689,-93.216,167.176,46.681,158.578
C08044=1025.599,-30.939,-93.203,167.172,46.684,158.578
C08045=1025.593,-31.188,-93.190,167.170,46.686,158.578
C08046=1025.588,-31.438,-93.178,167.167,46.689,158.578
C08047=1025.581,-31.688,-93.164,167.164,46.692,158.578
C08048=1025.575,-31.937,-93.152,167.161,46.695,158.578
C08049=1025.569,-32.187,-93.139,167.159,46.698,158.579
C08050=1025.563,-32.437,-93.126,167.156,46.701,158.579
C08051=1025.557,-32.687,-93.113,167.153,46.704,158.579
C08052=1025.551,-32.936,-93.100,167.150,46.706,158.579
C08053=1025.545,-33.186,-93.088,167.148,46.709,158.579
C08054=1025.539,-33.436,-93.075,167.144,46.712,158.579
C08055=1025.533,-33.685,-93.062,167.142,46.715,158.580
C08056=1025.527,-33.935,-93.049,167.139,46.718,158.580
C08057=1025.521,-34.184,-93.037,167.137,46.721,158.580
C08058=1025.514,-34.434,-93.024,167.133,46.723,158.580
C08059=1025.508,-34.683,-93.011,167.131,46.726,158.580
C08060=1025.503,-34.933,-92.999,167.128,46.729,158.580
C08061=1025.496,-35.183,-92.986,167.125,46.732,158.581
C08062=1025.491,-35.432,-92.973,167.122,46.735,158.581
C08063=1025.485,-35.682,-92.961,167.120,46.737,158.581
C08064=1025.479,-35.932,-92.948,167.116,46.740,158.581
C08065=1025.473,-36.181,-92.935,167.114,46.743,158.581
C08066=1025.466,-36.460,-92.922,167.111,46.746,158.581
C08067=1025.459,-36.741,-92.907,167.108,46.749,158.582
C08068=1025.453,-37.020,-92.893,167.104,46.752,158.582
C08069=1025.446,-37.300,-92.879,167.101,46.756,158.582
C08070=1025.441,-37.550,-92.867,167.098,46.758,158.582
C08071=1025.434,-37.799,-92.853,167.096,46.761,158.582
C08072=1025.428,-38.049,-92.841,167.092,46.764,158.582
C08073=1025.422,-38.299,-92.829,167.090,46.767,158.583
C08074=1025.416,-38.548,-92.816,167.086,46.769,158.583
C08075=1025.410,-38.798,-92.804,167.084,46.772,158.583
C08076=1025.404,-39.047,-92.791,167.081,46.775,158.583
C08077=1025.398,-39.297,-92.778,167.079,46.778,158.583
C08078=1025.392,-39.547,-92.766,167.076,46.781,158.583
C08079=1025.386,-39.796,-92.754,167.073,46.783,158.584
C08080=1025.380,-40.046,-92.741,167.070,46.787,158.584
C08081=1025.373,-40.296,-92.729,167.067,46.790,158.584
C08082=1025.367,-40.546,-92.717,167.064,46.792,158.584
C08083=1025.362,-40.795,-92.704,167.061,46.795,158.584
C08084=1025.355,-41.044,-92.692,167.059,46.798,158.584
C08085=1025.350,-41.294,-92.680,167.056,46.801,158.585
C08086=1025.344,-41.544,-92.667,167.053,46.803,158.585
C08087=1025.337,-41.794,-92.655,167.050,46.807,158.585
C08088=1025.332,-42.043,-92.643,167.047,46.810,158.585
C08089=1025.326,-42.293,-92.631,167.045,46.812,158.585
C08090=1025.319,-42.542,-92.619,167.041,46.815,158.585
C08091=1025.313,-42.792,-92.606,167.039,46.818,158.586
C08092=1025.307,-43.041,-92.595,167.036,46.821,158.586
C08093=1025.301,-43.291,-92.582,167.033,46.823,158.586
C08094=1025.295,-43.541,-92.569,167.030,46.827,158.586
C08095=1025.289,-43.790,-92.557,167.027,46.830,158.586
C08096=1025.283,-44.040,-92.545,167.025,46.832,158.586
C08097=1025.277,-44.289,-92.533,167.021,46.836,158.587
C08098=1025.271,-44.539,-92.521,167.019,46.838,158.587
C08099=1025.265,-44.789,-92.509,167.016,46.841,158.587
C08100=1025.259,-45.038,-92.497,167.013,46.844,158.587
C08101=1025.253,-45.288,-92.485,167.010,46.847,158.587
C08102=1025.247,-45.538,-92.472,167.007,46.850,158.587
C08103=1025.241,-45.788,-92.460,167.005,46.852,158.588
C08104=1025.235,-46.037,-92.448,167.001,46.856,158.588
C08105=1025.229,-46.286,-92.436,166.999,46.858,158.588
C08106=1025.223,-46.536,-92.424,166.996,46.861,158.588
C08107=1025.218,-46.786,-92.412,166.993,46.864,158.588
C08108=1025.211,-47.036,-92.400,166.990,46.867,158.588
C08109=1025.205,-47.286,-92.388,166.987,46.870,158.588
C08110=1025.199,-47.534,-92.376,166.985,46.873,158.589
C08111=1025.193,-47.784,-92.363,166.981,46.876,158.589
C08112=1025.187,-48.034,-92.351,166.979,46.878,158.589
C08113=1025.182,-48.284,-92.340,166.976,46.881,158.589
C08114=1025.176,-48.534,-92.327,166.972,46.884,158.589
C08115=1025.169,-48.783,-92.316,166.970,46.887,158.589
C08116=1025.164,-49.032,-92.303,166.967,46.890,158.590
C08117=1025.158,-49.283,-92.291,166.965,46.893,158.590
C08118=1025.152,-49.532,-92.280,166.961,46.896,158.590
C08119=1025.146,-49.782,-92.267,166.959,46.898,158.590
C08120=1025.140,-50.031,-92.255,166.956,46.901,158.590
C08121=1025.135,-50.281,-92.244,166.952,46.904,158.590
C08122=1025.129,-50.531,-92.231,166.950,46.907,158.591
C08123=1025.122,-50.780,-92.219,166.947,46.910,158.591
C08124=1025.117,-51.030,-92.208,166.945,46.913,158.591
C08125=1025.110,-51.280,-92.196,166.941,46.916,158.591
C08126=1025.104,-51.529,-92.184,166.938,46.919,158.591
C08127=1025.098,-51.779,-92.173,166.935,46.922,158.591
C08128=1025.091,-52.028,-92.161,166.933,46.925,158.592
C08129=1025.086,-52.278,-92.150,166.929,46.928,158.592
C08130=1025.078,-52.582,-92.136,166.926,46.932,158.592
C08131=1025.071,-52.886,-92.121,166.922,46.936,158.592
C08132=1025.064,-53.190,-92.108,166.919,46.939,158.592
C08133=1025.056,-53.494,-92.093,166.915,46.943,158.593
C08134=1025.050,-53.744,-92.082,166.912,46.946,158.593
C08135=1025.044,-53.993,-92.070,166.910,46.949,158.593
C08136=1025.038,-54.243,-92.059,166.906,46.952,158.593
C08137=1025.032,-54.492,-92.047,166.903,46.955,158.593
C08138=1025.026,-54.742,-92.036,166.901,46.958,158.594
C08139=1025.019,-54.992,-92.024,166.898,46.961,158.594
C08140=1025.013,-55.241,-92.013,166.894,46.964,158.594
C08141=1025.007,-55.491,-92.000,166.892,46.967,158.594
C08142=1025.002,-55.741,-91.989,166.889,46.970,158.594
C08143=1024.995,-55.991,-91.978,166.886,46.973,158.594
C08144=1024.989,-56.240,-91.967,166.883,46.976,158.595
C08145=1024.983,-56.490,-91.955,166.880,46.979,158.595
C08146=1024.978,-56.739,-91.943,166.877,46.982,158.595
C08147=1024.971,-56.989,-91.932,166.874,46.985,158.595
C08148=1024.966,-57.239,-91.921,166.872,46.988,158.595
C08149=1024.959,-57.489,-91.909,166.868,46.991,158.595
C08150=1024.953,-57.738,-91.898,166.865,46.994,158.596
C08151=1024.947,-57.988,-91.886,166.863,46.997,158.596
C08152=1024.942,-58.237,-91.875,166.860,47.000,158.596
C08153=1024.935,-58.488,-91.864,166.856,47.003,158.596
C08154=1024.929,-58.736,-91.852,166.854,47.006,158.596
C08155=1024.923,-58.987,-91.841,166.851,47.009,158.596
C08156=1024.917,-59.236,-91.830,166.848,47.012,158.597
C08157=1024.911,-59.487,-91.818,166.845,47.015,158.597
C08158=1024.905,-59.736,-91.806,166.842,47.018,158.597
C08159=1024.900,-59.985,-91.796,166.839,47.021,158.597
C08160=1024.893,-60.235,-91.784,166.837,47.024,158.597
C08161=1024.887,-60.484,-91.773,166.833,47.027,158.597
C08162=1024.881,-60.734,-91.761,166.830,47.030,158.598
C08163=1024.876,-60.984,-91.750,166.828,47.033,158.598
C08164=1024.870,-61.234,-91.739,166.825,47.036,158.598
C08165=1024.864,-61.483,-91.727,166.821,47.039,158.598
C08166=1024.858,-61.733,-91.716,166.818,47.042,158.598
C08167=1024.852,-61.983,-91.705,166.816,47.045,158.598
C08168=1024.846,-62.232,-91.694,166.813,47.048,158.599
C08169=1024.840,-62.481,-91.682,166.809,47.051,158.599
C08170=1024.834,-62.720,-91.671,166.807,47.054,158.599
C08171=1024.828,-62.958,-91.661,166.804,47.056,158.599
C08172=1024.823,-63.195,-91.651,166.801,47.059,158.599
C08173=1024.818,-63.434,-91.639,166.798,47.062,158.599
C08174=1024.812,-63.671,-91.629,166.796,47.065,158.600
C08175=1024.806,-63.909,-91.618,166.793,47.068,158.600
C08176=1024.801,-64.146,-91.607,166.790,47.070,158.600
C08177=1024.795,-64.384,-91.597,166.787,47.073,158.600
C08178=1024.789,-64.634,-91.586,166.785,47.076,158.600
///RCONF 1,0,0,1,0,0,0,0,0,0,0,0,0,0,0,0,0,0,0,0,0,0,0,0
C08179=1024.784,-64.883,-91.575,166.782,47.079,158.600
C08180=1024.777,-65.134,-91.564,166.778,47.082,158.600
C08181=1024.772,-65.383,-91.552,166.776,47.085,158.601
C08182=1024.766,-65.633,-91.541,166.773,47.088,158.601
C08183=1024.760,-65.882,-91.529,166.770,47.091,158.601
C08184=1024.754,-66.132,-91.518,166.767,47.093,158.601
C08185=1024.748,-66.381,-91.508,166.764,47.097,158.601
C08186=1024.742,-66.632,-91.496,166.761,47.100,158.601
C08187=1024.736,-66.881,-91.485,166.758,47.103,158.601
C08188=1024.730,-67.131,-91.475,166.755,47.106,158.602
C08189=1024.725,-67.380,-91.463,166.752,47.109,158.602
C08190=1024.719,-67.631,-91.452,166.750,47.112,158.602
C08191=1024.713,-67.880,-91.441,166.746,47.115,158.602
C08192=1024.708,-68.130,-91.430,166.743,47.118,158.602
C08193=1024.702,-68.379,-91.419,166.741,47.120,158.602
C08194=1024.696,-68.661,-91.407,166.737,47.124,158.602
C08195=1024.689,-68.942,-91.394,166.733,47.127,158.603
C08196=1024.682,-69.223,-91.382,166.730,47.130,158.603
C08197=1024.676,-69.505,-91.369,166.727,47.133,158.603
C08198=1024.670,-69.754,-91.359,166.724,47.136,158.603
C08199=1024.664,-70.005,-91.347,166.721,47.139,158.603
C08200=1024.658,-70.254,-91.336,166.718,47.142,158.603
C08201=1024.653,-70.504,-91.326,166.715,47.145,158.604
C08202=1024.647,-70.753,-91.315,166.713,47.148,158.604
C08203=1024.641,-71.003,-91.304,166.709,47.151,158.604
C08204=1024.636,-71.253,-91.292,166.706,47.154,158.604
C08205=1024.630,-71.503,-91.281,166.704,47.157,158.604
C08206=1024.624,-71.752,-91.270,166.700,47.160,158.604
C08207=1024.618,-72.002,-91.259,166.697,47.163,158.604
C08208=1024.613,-72.251,-91.248,166.695,47.166,158.605
C08209=1024.607,-72.501,-91.238,166.692,47.169,158.605
C08210=1024.601,-72.750,-91.227,166.688,47.171,158.605
C08211=1024.595,-73.001,-91.216,166.686,47.174,158.605
C08212=1024.589,-73.250,-91.205,166.683,47.177,158.605
C08213=1024.584,-73.500,-91.194,166.680,47.180,158.605
C08214=1024.579,-73.750,-91.183,166.677,47.183,158.605
C08215=1024.573,-73.999,-91.172,166.674,47.186,158.606
C08216=1024.567,-74.249,-91.161,166.671,47.189,158.605
C08217=1024.562,-74.499,-91.151,166.668,47.191,158.606
C08218=1024.555,-74.749,-91.140,166.665,47.195,158.606
C08219=1024.549,-74.998,-91.130,166.662,47.198,158.606
C08220=1024.543,-75.248,-91.119,166.659,47.201,158.606
C08221=1024.538,-75.498,-91.109,166.655,47.204,158.606
C08222=1024.532,-75.747,-91.098,166.653,47.207,158.606
C08223=1024.526,-75.997,-91.087,166.650,47.210,158.607
C08224=1024.520,-76.246,-91.077,166.647,47.213,158.607
C08225=1024.514,-76.496,-91.066,166.643,47.216,158.607
C08226=1024.509,-76.746,-91.056,166.641,47.219,158.607
C08227=1024.503,-76.996,-91.045,166.638,47.222,158.607
C08228=1024.497,-77.246,-91.034,166.635,47.225,158.607
C08229=1024.491,-77.496,-91.024,166.631,47.228,158.607
C08230=1024.485,-77.745,-91.014,166.629,47.231,158.608
C08231=1024.479,-77.995,-91.003,166.626,47.234,158.608
C08232=1024.474,-78.245,-90.993,166.623,47.237,158.608
C08233=1024.468,-78.494,-90.982,166.619,47.240,158.608
C08234=1024.462,-78.744,-90.972,166.617,47.243,158.608
C08235=1024.456,-78.993,-90.961,166.614,47.246,158.608
C08236=1024.451,-79.244,-90.951,166.611,47.249,158.609
C08237=1024.445,-79.493,-90.940,166.608,47.253,158.609
C08238=1024.439,-79.743,-90.930,166.605,47.255,158.609
C08239=1024.433,-79.992,-90.920,166.602,47.259,158.609
C08240=1024.428,-80.242,-90.910,166.599,47.262,158.609
C08241=1024.422,-80.492,-90.899,166.596,47.266,158.609
C08242=1024.416,-80.742,-90.889,166.594,47.268,158.610
C08243=1024.410,-80.991,-90.878,166.590,47.271,158.610
C08244=1024.404,-81.241,-90.869,166.587,47.275,158.610
C08245=1024.398,-81.490,-90.858,166.584,47.278,158.610
C08246=1024.392,-81.740,-90.848,166.581,47.281,158.610
C08247=1024.386,-81.990,-90.838,166.577,47.284,158.610
C08248=1024.380,-82.240,-90.828,166.576,47.288,158.611
C08249=1024.374,-82.490,-90.818,166.572,47.291,158.611
C08250=1024.368,-82.739,-90.808,166.569,47.294,158.611
C08251=1024.363,-82.989,-90.797,166.566,47.297,158.611
C08252=1024.356,-83.239,-90.788,166.563,47.300,158.611
C08253=1024.351,-83.489,-90.777,166.559,47.303,158.611
C08254=1024.344,-83.738,-90.767,166.557,47.306,158.612
C08255=1024.339,-83.988,-90.757,166.554,47.310,158.612
C08256=1024.333,-84.238,-90.747,166.551,47.313,158.612
C08257=1024.327,-84.487,-90.737,166.548,47.316,158.612
C08258=1024.320,-84.771,-90.726,166.544,47.319,158.612
C08259=1024.314,-85.055,-90.714,166.540,47.323,158.612
C08260=1024.308,-85.337,-90.703,166.537,47.326,158.613
C08261=1024.301,-85.621,-90.691,166.534,47.330,158.613
C08262=1024.295,-85.871,-90.682,166.531,47.333,158.613
C08263=1024.290,-86.121,-90.671,166.528,47.336,158.613
C08264=1024.283,-86.370,-90.661,166.525,47.340,158.613
C08265=1024.278,-86.620,-90.651,166.522,47.342,158.613
C08266=1024.272,-86.870,-90.641,166.519,47.346,158.614
C08267=1024.266,-87.120,-90.631,166.516,47.349,158.614
C08268=1024.260,-87.370,-90.622,166.513,47.352,158.614
C08269=1024.255,-87.619,-90.611,166.510,47.356,158.614
C08270=1024.249,-87.869,-90.602,166.506,47.359,158.614
C08271=1024.243,-88.119,-90.591,166.504,47.362,158.614
C08272=1024.237,-88.369,-90.582,166.501,47.365,158.615
C08273=1024.232,-88.619,-90.572,166.498,47.368,158.615
C08274=1024.225,-88.868,-90.561,166.495,47.371,158.615
C08275=1024.220,-89.117,-90.552,166.491,47.374,158.615
C08276=1024.214,-89.367,-90.542,166.489,47.377,158.615
C08277=1024.209,-89.617,-90.532,166.486,47.380,158.615
C08278=1024.203,-89.867,-90.522,166.483,47.384,158.616
C08279=1024.197,-90.117,-90.512,166.480,47.387,158.616
C08280=1024.192,-90.366,-90.503,166.476,47.390,158.616
C08281=1024.185,-90.616,-90.493,166.474,47.393,158.616
C08282=1024.180,-90.866,-90.483,166.471,47.396,158.616
C08283=1024.174,-91.115,-90.473,166.468,47.399,158.616
C08284=1024.169,-91.365,-90.463,166.464,47.402,158.616
C08285=1024.163,-91.614,-90.454,166.461,47.406,158.616
C08286=1024.157,-91.865,-90.443,166.459,47.408,158.617
C08287=1024.151,-92.114,-90.434,166.456,47.412,158.617
C08288=1024.146,-92.364,-90.424,166.453,47.415,158.617
C08289=1024.140,-92.614,-90.415,166.449,47.418,158.617
C08290=1024.135,-92.864,-90.404,166.446,47.421,158.617
C08291=1024.128,-93.113,-90.395,166.444,47.424,158.617
C08292=1024.124,-93.363,-90.385,166.441,47.427,158.618
C08293=1024.117,-93.613,-90.375,166.437,47.430,158.618
C08294=1024.112,-93.863,-90.365,166.434,47.433,158.618
C08295=1024.106,-94.113,-90.356,166.431,47.436,158.618
C08296=1024.101,-94.362,-90.346,166.429,47.439,158.618
C08297=1024.095,-94.612,-90.336,166.426,47.443,158.618
C08298=1024.089,-94.862,-90.327,166.423,47.446,158.619
C08299=1024.084,-95.111,-90.317,166.419,47.449,158.619
C08300=1024.078,-95.361,-90.307,166.416,47.452,158.619
C08301=1024.072,-95.611,-90.297,166.414,47.455,158.619
C08302=1024.067,-95.860,-90.288,166.411,47.458,158.619
C08303=1024.061,-96.111,-90.279,166.407,47.462,158.619
C08304=1024.055,-96.361,-90.269,166.404,47.465,158.619
C08305=1024.050,-96.610,-90.259,166.401,47.468,158.619
C08306=1024.044,-96.860,-90.250,166.399,47.471,158.620
C08307=1024.039,-97.109,-90.240,166.395,47.474,158.620
C08308=1024.033,-97.359,-90.230,166.392,47.477,158.620
C08309=1024.027,-97.609,-90.221,166.389,47.480,158.620
C08310=1024.022,-97.858,-90.211,166.386,47.483,158.620
C08311=1024.016,-98.109,-90.202,166.384,47.486,158.620
C08312=1024.010,-98.358,-90.193,166.380,47.489,158.620
C08313=1024.005,-98.607,-90.183,166.377,47.492,158.621
C08314=1023.998,-98.857,-90.174,166.374,47.496,158.621
C08315=1023.994,-99.107,-90.165,166.371,47.499,158.621
C08316=1023.988,-99.357,-90.155,166.368,47.503,158.621
C08317=1023.982,-99.607,-90.146,166.364,47.506,158.621
C08318=1023.976,-99.857,-90.137,166.361,47.509,158.621
C08319=1023.970,-100.106,-90.127,166.359,47.512,158.622
C08320=1023.965,-100.355,-90.118,166.356,47.516,158.622
C08321=1023.959,-100.606,-90.109,166.353,47.519,158.622
C08322=1023.952,-100.891,-90.098,166.349,47.523,158.622
C08323=1023.946,-101.177,-90.088,166.346,47.526,158.622
C08324=1023.940,-101.462,-90.076,166.343,47.530,158.623
C08325=1023.933,-101.748,-90.067,166.338,47.533,158.623
C08326=1023.928,-101.999,-90.057,166.335,47.537,158.623
C08327=1023.922,-102.248,-90.048,166.332,47.540,158.623
C08328=1023.916,-102.498,-90.038,166.330,47.543,158.623
C08329=1023.911,-102.747,-90.030,166.327,47.546,158.623
C08330=1023.905,-102.997,-90.020,166.324,47.549,158.623
C08331=1023.899,-103.247,-90.012,166.320,47.553,158.623
C08332=1023.893,-103.497,-90.002,166.317,47.556,158.624
C08333=1023.888,-103.746,-89.992,166.314,47.560,158.624
C08334=1023.883,-103.996,-89.984,166.311,47.563,158.624
C08335=1023.877,-104.246,-89.974,166.309,47.566,158.624
C08336=1023.871,-104.496,-89.966,166.306,47.569,158.624
C08337=1023.866,-104.745,-89.956,166.302,47.572,158.624
C08338=1023.860,-104.995,-89.948,166.299,47.576,158.625
C08339=1023.854,-105.245,-89.938,166.296,47.579,158.625
C08340=1023.849,-105.495,-89.929,166.293,47.582,158.625
C08341=1023.843,-105.744,-89.920,166.290,47.585,158.625
C08342=1023.838,-105.995,-89.911,166.287,47.588,158.625
C08343=1023.832,-106.244,-89.902,166.284,47.591,158.625
C08344=1023.826,-106.494,-89.893,166.281,47.595,158.626
C08345=1023.820,-106.743,-89.884,166.278,47.598,158.626
C08346=1023.815,-106.993,-89.875,166.275,47.601,158.626
C08347=1023.809,-107.244,-89.866,166.272,47.605,158.626
C08348=1023.804,-107.493,-89.857,166.268,47.608,158.626
C08349=1023.798,-107.743,-89.848,166.265,47.611,158.626
C08350=1023.792,-107.992,-89.839,166.263,47.614,158.627
C08351=1023.786,-108.243,-89.830,166.260,47.618,158.627
C08352=1023.781,-108.492,-89.822,166.257,47.621,158.627
C08353=1023.776,-108.741,-89.812,166.254,47.624,158.627
C08354=1023.770,-108.992,-89.804,166.251,47.628,158.627
C08355=1023.765,-109.242,-89.795,166.247,47.631,158.627
C08356=1023.758,-109.491,-89.786,166.244,47.634,158.627
C08357=1023.753,-109.741,-89.777,166.241,47.637,158.628
C08358=1023.748,-109.991,-89.769,166.238,47.641,158.628
C08359=1023.742,-110.241,-89.759,166.236,47.644,158.628
C08360=1023.736,-110.490,-89.751,166.233,47.647,158.628
C08361=1023.731,-110.740,-89.742,166.229,47.650,158.628
C08362=1023.725,-110.990,-89.733,166.226,47.654,158.629
C08363=1023.720,-111.239,-89.724,166.223,47.657,158.629
C08364=1023.714,-111.489,-89.716,166.220,47.661,158.629
C08365=1023.708,-111.739,-89.707,166.217,47.664,158.629
C08366=1023.703,-111.989,-89.699,166.214,47.668,158.629
C08367=1023.697,-112.238,-89.690,166.211,47.671,158.629
C08368=1023.691,-112.489,-89.681,166.208,47.674,158.629
C08369=1023.686,-112.738,-89.672,166.205,47.677,158.630
C08370=1023.681,-112.988,-89.664,166.202,47.680,158.630
C08371=1023.675,-113.238,-89.655,166.199,47.684,158.630
C08372=1023.669,-113.487,-89.646,166.196,47.687,158.630
C08373=1023.664,-113.737,-89.637,166.192,47.690,158.630
C08374=1023.658,-113.988,-89.628,166.189,47.693,158.630
C08375=1023.653,-114.237,-89.620,166.186,47.697,158.631
C08376=1023.647,-114.487,-89.611,166.183,47.700,158.631
C08377=1023.641,-114.736,-89.603,166.181,47.703,158.631
C08378=1023.636,-114.987,-89.595,166.178,47.706,158.631
C08379=1023.630,-115.237,-89.586,166.175,47.710,158.631
C08380=1023.625,-115.486,-89.578,166.171,47.713,158.631
C08381=1023.620,-115.735,-89.568,166.168,47.717,158.631
C08382=1023.613,-115.985,-89.560,166.165,47.720,158.632
C08383=1023.608,-116.235,-89.552,166.162,47.724,158.632
C08384=1023.602,-116.485,-89.543,166.159,47.727,158.632
C08385=1023.597,-116.735,-89.535,166.156,47.730,158.632
C08386=1023.590,-117.020,-89.525,166.153,47.734,158.632
C08387=1023.584,-117.306,-89.516,166.149,47.738,158.632
C08388=1023.577,-117.591,-89.506,166.146,47.742,158.633
C08389=1023.571,-117.876,-89.497,166.142,47.745,158.633
C08390=1023.566,-118.126,-89.488,166.140,47.749,158.633
C08391=1023.561,-118.376,-89.480,166.136,47.752,158.633
C08392=1023.555,-118.625,-89.471,166.133,47.755,158.633
C08393=1023.549,-118.875,-89.463,166.130,47.759,158.634
C08394=1023.544,-119.125,-89.454,166.127,47.762,158.634
C08395=1023.538,-119.375,-89.446,166.124,47.765,158.634
C08396=1023.533,-119.625,-89.437,166.121,47.769,158.634
C08397=1023.527,-119.874,-89.429,166.118,47.772,158.634
C08398=1023.522,-120.124,-89.422,166.114,47.776,158.634
C08399=1023.516,-120.375,-89.413,166.111,47.779,158.634
C08400=1023.510,-120.624,-89.405,166.108,47.783,158.635
C08401=1023.505,-120.874,-89.396,166.106,47.786,158.635
C08402=1023.500,-121.124,-89.388,166.103,47.789,158.635
C08403=1023.494,-121.373,-89.380,166.100,47.792,158.635
C08404=1023.488,-121.623,-89.372,166.097,47.796,158.635
C08405=1023.483,-121.873,-89.364,166.094,47.799,158.635
C08406=1023.478,-122.123,-89.355,166.090,47.802,158.636
C08407=1023.472,-122.373,-89.347,166.087,47.806,158.636
C08408=1023.466,-122.623,-89.339,166.084,47.809,158.636
C08409=1023.461,-122.872,-89.330,166.081,47.812,158.636
C08410=1023.455,-123.122,-89.322,166.078,47.816,158.636
C08411=1023.450,-123.372,-89.314,166.076,47.819,158.636
C08412=1023.445,-123.622,-89.306,166.073,47.822,158.637
C08413=1023.439,-123.871,-89.298,166.069,47.826,158.637
C08414=1023.434,-124.121,-89.290,166.066,47.829,158.637
C08415=1023.429,-124.371,-89.282,166.063,47.833,158.637
C08416=1023.423,-124.621,-89.274,166.060,47.836,158.637
C08417=1023.417,-124.870,-89.265,166.057,47.840,158.637
C08418=1023.412,-125.121,-89.258,166.054,47.843,158.637
C08419=1023.406,-125.370,-89.250,166.051,47.846,158.638
C08420=1023.401,-125.620,-89.241,166.048,47.850,158.638
C08421=1023.395,-125.870,-89.234,166.044,47.853,158.638
///RCONF 1,0,0,0,0,0,0,0,0,0,0,0,0,0,0,0,0,0,0,0,0,0,0,0
C08422=1023.390,-126.119,-89.226,166.042,47.857,158.638
C08423=1023.384,-126.369,-89.218,166.038,47.860,158.638
C08424=1023.379,-126.619,-89.210,166.036,47.863,158.639
C08425=1023.373,-126.869,-89.202,166.033,47.867,158.639
C08426=1023.368,-127.118,-89.194,166.030,47.870,158.639
C08427=1023.362,-127.368,-89.186,166.027,47.873,158.639
C08428=1023.357,-127.618,-89.178,166.024,47.877,158.639
C08429=1023.351,-127.868,-89.171,166.021,47.880,158.639
C08430=1023.346,-128.118,-89.162,166.017,47.884,158.639
C08431=1023.341,-128.368,-89.153,166.015,47.886,158.640
C08432=1023.337,-128.617,-89.144,166.012,47.889,158.640
C08433=1023.333,-128.867,-89.134,166.009,47.890,158.639
C08434=1023.331,-129.116,-89.124,166.006,47.892,158.639
C08435=1023.327,-129.366,-89.113,166.004,47.892,158.639
C08436=1023.325,-129.616,-89.101,166.002,47.892,158.639
C08437=1023.324,-129.865,-89.089,165.999,47.892,158.638
C08438=1023.323,-130.115,-89.076,165.997,47.891,158.638
C08439=1023.321,-130.365,-89.062,165.994,47.890,158.637
C08440=1023.321,-130.615,-89.048,165.992,47.888,158.637
C08441=1023.322,-130.864,-89.034,165.990,47.886,158.636
C08442=1023.323,-131.114,-89.020,165.987,47.883,158.635
C08443=1023.324,-131.364,-89.004,165.986,47.880,158.635
C08444=1023.325,-131.614,-88.987,165.984,47.876,158.634
C08445=1023.329,-131.864,-88.971,165.983,47.872,158.633
C08446=1023.332,-132.114,-88.952,165.981,47.867,158.632
C08447=1023.335,-132.364,-88.935,165.980,47.862,158.631
C08448=1023.339,-132.613,-88.916,165.978,47.856,158.630
C08449=1023.343,-132.863,-88.897,165.977,47.850,158.628
C08450=1023.051,-132.889,-89.238,165.929,48.138,158.670
C08451=1023.046,-132.639,-89.258,165.930,48.144,158.671
C08452=1023.042,-132.390,-89.275,165.931,48.150,158.673
C08453=1023.039,-132.139,-89.294,165.934,48.155,158.674
C08454=1023.036,-131.890,-89.311,165.934,48.160,158.675
C08455=1023.034,-131.640,-89.329,165.936,48.164,158.676
C08456=1023.031,-131.390,-89.345,165.938,48.168,158.676
C08457=1023.030,-131.140,-89.360,165.940,48.171,158.677
C08458=1023.030,-130.891,-89.375,165.943,48.174,158.678
C08459=1023.029,-130.640,-89.390,165.945,48.176,158.679
C08460=1023.030,-130.391,-89.404,165.947,48.178,158.680
C08461=1023.030,-130.141,-89.418,165.949,48.179,158.680
C08462=1023.031,-129.891,-89.430,165.951,48.180,158.680
C08463=1023.032,-129.642,-89.442,165.954,48.180,158.681
C08464=1023.035,-129.392,-89.454,165.956,48.180,158.681
C08465=1023.037,-129.142,-89.465,165.959,48.179,158.681
C08466=1023.041,-128.893,-89.475,165.962,48.178,158.681
C08467=1023.044,-128.643,-89.486,165.965,48.176,158.682
C08468=1023.048,-128.393,-89.495,165.967,48.174,158.682
C08469=1023.053,-128.144,-89.503,165.971,48.171,158.682
C08470=1023.058,-127.894,-89.512,165.973,48.168,158.681
C08471=1023.064,-127.644,-89.520,165.976,48.164,158.681
C08472=1023.069,-127.394,-89.527,165.979,48.161,158.681
C08473=1023.075,-127.145,-89.536,165.982,48.157,158.681
C08474=1023.080,-126.895,-89.543,165.985,48.154,158.681
C08475=1023.086,-126.645,-89.551,165.988,48.150,158.680
C08476=1023.092,-126.396,-89.559,165.991,48.147,158.680
C08477=1023.097,-126.145,-89.567,165.994,48.144,158.680
C08478=1023.103,-125.896,-89.575,165.997,48.140,158.680
C08479=1023.108,-125.646,-89.583,166.000,48.137,158.680
C08480=1023.114,-125.396,-89.591,166.003,48.133,158.680
C08481=1023.119,-125.146,-89.599,166.006,48.130,158.680
C08482=1023.124,-124.896,-89.607,166.010,48.126,158.679
C08483=1023.130,-124.647,-89.615,166.013,48.122,158.679
C08484=1023.135,-124.397,-89.623,166.016,48.119,158.679
C08485=1023.141,-124.147,-89.630,166.019,48.115,158.679
C08486=1023.146,-123.897,-89.639,166.022,48.112,158.679
C08487=1023.151,-123.647,-89.647,166.025,48.109,158.679
C08488=1023.157,-123.398,-89.655,166.028,48.105,158.678
C08489=1023.162,-123.148,-89.663,166.031,48.102,158.678
C08490=1023.167,-122.898,-89.672,166.034,48.099,158.678
C08491=1023.173,-122.649,-89.679,166.036,48.095,158.678
C08492=1023.179,-122.399,-89.688,166.039,48.092,158.678
C08493=1023.184,-122.149,-89.696,166.043,48.089,158.678
C08494=1023.189,-121.899,-89.704,166.046,48.085,158.677
C08495=1023.196,-121.649,-89.712,166.049,48.081,158.677
C08496=1023.201,-121.399,-89.721,166.052,48.078,158.677
C08497=1023.206,-121.149,-89.729,166.055,48.074,158.677
C08498=1023.212,-120.900,-89.737,166.058,48.071,158.677
C08499=1023.217,-120.650,-89.745,166.061,48.067,158.677
C08500=1023.222,-120.400,-89.754,166.064,48.064,158.676
C08501=1023.228,-120.150,-89.762,166.067,48.061,158.676
C08502=1023.234,-119.901,-89.770,166.070,48.057,158.676
C08503=1023.239,-119.651,-89.778,166.074,48.054,158.676
C08504=1023.245,-119.401,-89.787,166.077,48.051,158.676
C08505=1023.251,-119.151,-89.795,166.080,48.047,158.676
C08506=1023.256,-118.901,-89.804,166.083,48.043,158.676
C08507=1023.261,-118.652,-89.812,166.086,48.040,158.675
C08508=1023.267,-118.402,-89.821,166.089,48.036,158.675
C08509=1023.272,-118.152,-89.828,166.092,48.033,158.675
C08510=1023.278,-117.902,-89.837,166.094,48.030,158.675
C08511=1023.284,-117.617,-89.846,166.098,48.026,158.675
C08512=1023.291,-117.332,-89.856,166.101,48.022,158.674
C08513=1023.297,-117.047,-89.865,166.105,48.018,158.674
C08514=1023.303,-116.761,-89.876,166.108,48.014,158.674
C08515=1023.309,-116.512,-89.884,166.111,48.011,158.674
C08516=1023.314,-116.262,-89.892,166.114,48.008,158.674
C08517=1023.319,-116.012,-89.901,166.117,48.004,158.673
C08518=1023.325,-115.762,-89.909,166.121,48.001,158.673
C08519=1023.331,-115.512,-89.918,166.124,47.997,158.673
C08520=1023.337,-115.263,-89.926,166.127,47.994,158.673
C08521=1023.342,-115.013,-89.934,166.130,47.990,158.673
C08522=1023.348,-114.763,-89.943,166.133,47.986,158.673
C08523=1023.353,-114.513,-89.952,166.136,47.983,158.673
C08524=1023.358,-114.263,-89.960,166.139,47.980,158.672
C08525=1023.364,-114.013,-89.969,166.142,47.977,158.672
C08526=1023.370,-113.763,-89.977,166.145,47.973,158.672
C08527=1023.376,-113.514,-89.986,166.149,47.970,158.672
C08528=1023.381,-113.264,-89.995,166.152,47.967,158.672
C08529=1023.386,-113.015,-90.003,166.155,47.963,158.672
C08530=1023.392,-112.764,-90.012,166.157,47.960,158.671
C08531=1023.397,-112.515,-90.020,166.160,47.957,158.671
C08532=1023.403,-112.265,-90.029,166.163,47.953,158.671
C08533=1023.409,-112.015,-90.038,166.166,47.950,158.671
C08534=1023.414,-111.765,-90.047,166.169,47.946,158.671
C08535=1023.419,-111.516,-90.055,166.173,47.943,158.671
C08536=1023.425,-111.265,-90.064,166.176,47.939,158.670
C08537=1023.431,-111.016,-90.073,166.179,47.936,158.670
C08538=1023.436,-110.766,-90.082,166.182,47.933,158.670
C08539=1023.442,-110.516,-90.091,166.185,47.930,158.670
C08540=1023.448,-110.267,-90.099,166.188,47.926,158.670
C08541=1023.453,-110.018,-90.108,166.191,47.923,158.670
C08542=1023.459,-109.767,-90.117,166.195,47.919,158.670
C08543=1023.465,-109.517,-90.125,166.197,47.916,158.669
C08544=1023.470,-109.268,-90.134,166.201,47.912,158.669
C08545=1023.476,-109.018,-90.143,166.203,47.910,158.669
C08546=1023.481,-108.768,-90.152,166.206,47.906,158.669
C08547=1023.487,-108.518,-90.160,166.209,47.902,158.669
C08548=1023.493,-108.269,-90.170,166.212,47.899,158.669
C08549=1023.498,-108.019,-90.178,166.215,47.895,158.668
C08550=1023.504,-107.769,-90.187,166.218,47.892,158.668
C08551=1023.509,-107.519,-90.196,166.221,47.889,158.668
C08552=1023.515,-107.270,-90.205,166.225,47.886,158.668
C08553=1023.521,-107.019,-90.214,166.228,47.882,158.668
C08554=1023.526,-106.770,-90.223,166.231,47.879,158.668
C08555=1023.532,-106.520,-90.232,166.234,47.876,158.667
C08556=1023.538,-106.271,-90.241,166.237,47.872,158.667
C08557=1023.543,-106.020,-90.250,166.240,47.869,158.667
C08558=1023.548,-105.771,-90.260,166.242,47.866,158.667
C08559=1023.554,-105.521,-90.268,166.246,47.862,158.667
C08560=1023.559,-105.271,-90.277,166.249,47.859,158.667
C08561=1023.565,-105.022,-90.286,166.252,47.855,158.666
C08562=1023.571,-104.771,-90.295,166.255,47.852,158.666
C08563=1023.576,-104.522,-90.304,166.258,47.849,158.666
C08564=1023.582,-104.272,-90.313,166.261,47.846,158.666
C08565=1023.588,-104.023,-90.322,166.264,47.842,158.666
C08566=1023.593,-103.772,-90.332,166.267,47.839,158.666
C08567=1023.599,-103.523,-90.341,166.271,47.836,158.666
C08568=1023.605,-103.273,-90.350,166.273,47.833,158.665
C08569=1023.610,-103.023,-90.359,166.276,47.830,158.665
C08570=1023.616,-102.773,-90.369,166.279,47.826,158.665
C08571=1023.621,-102.524,-90.377,166.282,47.823,158.665
C08572=1023.628,-102.274,-90.387,166.285,47.819,158.665
C08573=1023.632,-102.024,-90.396,166.289,47.816,158.665
C08574=1023.638,-101.774,-90.405,166.292,47.812,158.664
C08575=1023.645,-101.489,-90.415,166.295,47.809,158.664
C08576=1023.652,-101.203,-90.426,166.299,47.805,158.664
C08577=1023.658,-100.917,-90.437,166.302,47.801,158.664
C08578=1023.665,-100.632,-90.447,166.306,47.798,158.664
C08579=1023.669,-100.382,-90.457,166.309,47.794,158.663
C08580=1023.676,-100.133,-90.466,166.312,47.791,158.663
C08581=1023.681,-99.883,-90.475,166.314,47.788,158.663
C08582=1023.687,-99.633,-90.484,166.317,47.785,158.663
C08583=1023.693,-99.383,-90.494,166.320,47.781,158.663
C08584=1023.699,-99.134,-90.503,166.324,47.778,158.663
C08585=1023.704,-98.883,-90.512,166.327,47.774,158.663
C08586=1023.709,-98.634,-90.522,166.330,47.771,158.662
C08587=1023.716,-98.385,-90.531,166.333,47.767,158.662
C08588=1023.721,-98.135,-90.540,166.336,47.764,158.662
C08589=1023.727,-97.885,-90.549,166.339,47.761,158.662
C08590=1023.732,-97.635,-90.559,166.343,47.758,158.662
C08591=1023.738,-97.386,-90.569,166.344,47.754,158.661
C08592=1023.744,-97.136,-90.578,166.348,47.751,158.661
C08593=1023.749,-96.885,-90.588,166.351,47.748,158.661
C08594=1023.755,-96.636,-90.597,166.354,47.745,158.661
C08595=1023.760,-96.386,-90.607,166.357,47.742,158.661
C08596=1023.766,-96.137,-90.616,166.361,47.738,158.661
C08597=1023.771,-95.887,-90.626,166.363,47.736,158.661
C08598=1023.777,-95.637,-90.636,166.366,47.732,158.661
C08599=1023.782,-95.388,-90.646,166.369,47.729,158.660
C08600=1023.788,-95.138,-90.655,166.372,47.726,158.660
C08601=1023.794,-94.888,-90.665,166.376,47.723,158.660
C08602=1023.799,-94.639,-90.675,166.379,47.719,158.660
C08603=1023.805,-94.388,-90.683,166.382,47.716,158.660
C08604=1023.811,-94.138,-90.694,166.384,47.713,158.660
C08605=1023.816,-93.889,-90.703,166.387,47.710,158.659
C08606=1023.822,-93.639,-90.713,166.390,47.707,158.659
C08607=1023.828,-93.389,-90.723,166.394,47.703,158.659
C08608=1023.833,-93.140,-90.732,166.397,47.700,158.659
C08609=1023.839,-92.890,-90.742,166.400,47.697,158.659
C08610=1023.844,-92.640,-90.752,166.402,47.694,158.659
C08611=1023.851,-92.390,-90.762,166.405,47.690,158.659
C08612=1023.855,-92.141,-90.771,166.408,47.687,158.658
C08613=1023.862,-91.891,-90.781,166.412,47.684,158.658
C08614=1023.867,-91.641,-90.791,166.415,47.681,158.658
C08615=1023.873,-91.392,-90.800,166.418,47.678,158.658
C08616=1023.879,-91.142,-90.810,166.421,47.675,158.658
C08617=1023.884,-90.892,-90.821,166.423,47.672,158.658
C08618=1023.891,-90.643,-90.830,166.427,47.669,158.658
C08619=1023.896,-90.393,-90.840,166.430,47.665,158.657
C08620=1023.902,-90.143,-90.850,166.433,47.662,158.657
C08621=1023.907,-89.893,-90.860,166.436,47.658,158.657
C08622=1023.913,-89.643,-90.869,166.439,47.655,158.657
C08623=1023.919,-89.393,-90.880,166.441,47.652,158.657
C08624=1023.924,-89.144,-90.889,166.445,47.649,158.657
C08625=1023.930,-88.894,-90.899,166.448,47.646,158.656
C08626=1023.936,-88.644,-90.909,166.451,47.642,158.656
C08627=1023.942,-88.395,-90.919,166.454,47.639,158.656
C08628=1023.948,-88.145,-90.929,166.457,47.636,158.656
C08629=1023.953,-87.896,-90.939,166.461,47.633,158.656
C08630=1023.959,-87.646,-90.948,166.463,47.630,158.656
C08631=1023.964,-87.396,-90.959,166.466,47.627,158.656
C08632=1023.970,-87.146,-90.968,166.469,47.623,158.655
C08633=1023.976,-86.896,-90.979,166.472,47.620,158.655
C08634=1023.982,-86.647,-90.989,166.475,47.617,158.655
C08635=1023.988,-86.397,-90.999,166.479,47.613,158.655
C08636=1023.993,-86.147,-91.008,166.482,47.610,158.655
C08637=1023.999,-85.897,-91.018,166.485,47.606,158.654
C08638=1024.005,-85.648,-91.028,166.487,47.604,158.654
C08639=1024.011,-85.364,-91.040,166.491,47.600,158.654
C08640=1024.018,-85.081,-91.051,166.494,47.596,158.654
C08641=1024.025,-84.798,-91.063,166.498,47.592,158.654
C08642=1024.032,-84.514,-91.074,166.501,47.589,158.654
C08643=1024.037,-84.265,-91.083,166.504,47.586,158.653
C08644=1024.043,-84.014,-91.093,166.507,47.582,158.653
C08645=1024.049,-83.765,-91.104,166.511,47.579,158.653
C08646=1024.054,-83.515,-91.114,166.513,47.576,158.653
C08647=1024.061,-83.265,-91.123,166.516,47.573,158.653
C08648=1024.066,-83.016,-91.134,166.519,47.569,158.652
C08649=1024.073,-82.766,-91.144,166.522,47.566,158.652
C08650=1024.078,-82.516,-91.154,166.525,47.563,158.652
C08651=1024.084,-82.267,-91.164,166.529,47.560,158.652
C08652=1024.090,-82.017,-91.175,166.532,47.556,158.652
C08653=1024.096,-81.767,-91.184,166.534,47.553,158.652
C08654=1024.102,-81.517,-91.195,166.537,47.550,158.651
C08655=1024.107,-81.267,-91.205,166.540,47.547,158.651
C08656=1024.113,-81.018,-91.215,166.543,47.543,158.651
C08657=1024.119,-80.768,-91.226,166.546,47.540,158.651
C08658=1024.125,-80.518,-91.235,166.550,47.536,158.651
C08659=1024.131,-80.269,-91.246,166.553,47.533,158.651
C08660=1024.137,-80.019,-91.256,166.556,47.530,158.651
C08661=1024.143,-79.769,-91.266,166.558,47.527,158.650
C08662=1024.148,-79.519,-91.277,166.561,47.524,158.650
C08663=1024.154,-79.270,-91.288,166.565,47.521,158.650
C08664=1024.160,-79.020,-91.297,166.568,47.518,158.650
C08665=1024.166,-78.771,-91.308,166.571,47.515,158.650
C08666=1024.171,-78.520,-91.318,166.573,47.511,158.649
C08667=1024.177,-78.271,-91.329,166.576,47.508,158.649
C08668=1024.183,-78.021,-91.339,166.579,47.505,158.649
C08669=1024.189,-77.772,-91.349,166.583,47.502,158.649
C08670=1024.195,-77.522,-91.360,166.586,47.499,158.649
C08671=1024.200,-77.272,-91.370,166.588,47.496,158.649
C08672=1024.206,-77.023,-91.381,166.591,47.493,158.649
C08673=1024.211,-76.772,-91.392,166.595,47.490,158.648
C08674=1024.218,-76.523,-91.402,166.598,47.486,158.648
C08675=1024.224,-76.274,-91.413,166.601,47.483,158.648
C08676=1024.229,-76.024,-91.423,166.603,47.480,158.648
C08677=1024.235,-75.774,-91.434,166.606,47.477,158.648
C08678=1024.241,-75.524,-91.445,166.609,47.473,158.648
C08679=1024.247,-75.274,-91.455,166.613,47.470,158.647
C08680=1024.253,-75.025,-91.465,166.616,47.467,158.647
C08681=1024.259,-74.775,-91.476,166.618,47.464,158.647
C08682=1024.264,-74.525,-91.486,166.621,47.461,158.647
C08683=1024.270,-74.276,-91.497,166.625,47.458,158.647
C08684=1024.276,-74.026,-91.508,166.628,47.455,158.647
C08685=1024.281,-73.776,-91.518,166.630,47.452,158.646
C08686=1024.288,-73.526,-91.530,166.633,47.449,158.646
C08687=1024.293,-73.276,-91.540,166.636,47.446,158.646
C08688=1024.299,-73.027,-91.551,166.640,47.443,158.646
C08689=1024.305,-72.777,-91.562,166.642,47.440,158.646
C08690=1024.310,-72.528,-91.573,166.645,47.437,158.646
C08691=1024.315,-72.277,-91.584,166.649,47.434,158.646
C08692=1024.321,-72.028,-91.595,166.651,47.431,158.646
C08693=1024.327,-71.779,-91.606,166.654,47.428,158.645
C08694=1024.333,-71.528,-91.617,166.657,47.425,158.645
C08695=1024.339,-71.279,-91.628,166.660,47.422,158.645
C08696=1024.344,-71.029,-91.639,166.663,47.419,158.645
C08697=1024.350,-70.780,-91.650,166.666,47.416,158.645
C08698=1024.356,-70.530,-91.660,166.669,47.413,158.645
C08699=1024.362,-70.281,-91.671,166.671,47.410,158.644
C08700=1024.368,-70.031,-91.683,166.675,47.407,158.644
C08701=1024.373,-69.781,-91.694,166.678,47.404,158.644
C08702=1024.379,-69.531,-91.705,166.681,47.401,158.644
C08703=1024.386,-69.250,-91.717,166.684,47.397,158.644
C08704=1024.392,-68.969,-91.729,166.688,47.394,158.644
C08705=1024.398,-68.687,-91.742,166.690,47.390,158.644
C08706=1024.405,-68.406,-91.754,166.694,47.387,158.643
C08707=1024.411,-68.156,-91.765,166.697,47.384,158.643
C08708=1024.417,-67.907,-91.776,166.700,47.381,158.643
C08709=1024.422,-67.657,-91.787,166.702,47.378,158.643
C08710=1024.427,-67.408,-91.798,166.706,47.375,158.643
C08711=1024.434,-67.157,-91.809,166.709,47.372,158.643
C08712=1024.440,-66.908,-91.820,166.712,47.369,158.643
C08713=1024.445,-66.658,-91.831,166.714,47.366,158.642
C08714=1024.451,-66.409,-91.842,166.717,47.363,158.642
C08715=1024.457,-66.159,-91.853,166.721,47.360,158.642
C08716=1024.463,-65.909,-91.864,166.724,47.357,158.642
C08717=1024.468,-65.659,-91.876,166.726,47.354,158.642
C08718=1024.474,-65.409,-91.887,166.729,47.351,158.642
C08719=1024.481,-65.160,-91.898,166.733,47.348,158.641
C08720=1024.486,-64.911,-91.909,166.735,47.345,158.641
C08721=1024.492,-64.661,-91.920,166.738,47.342,158.641
C08722=1024.498,-64.411,-91.931,166.741,47.338,158.641
///RCONF 1,0,0,1,0,0,0,0,0,0,0,0,0,0,0,0,0,0,0,0,0,0,0,0
C08723=1024.504,-64.162,-91.942,166.744,47.335,158.641
C08724=1024.509,-63.912,-91.954,166.747,47.332,158.641
C08725=1024.515,-63.662,-91.965,166.750,47.329,158.640
C08726=1024.521,-63.412,-91.976,166.753,47.326,158.640
C08727=1024.527,-63.163,-91.987,166.756,47.323,158.640
C08728=1024.534,-62.913,-91.999,166.759,47.320,158.640
C08729=1024.539,-62.664,-92.010,166.762,47.317,158.640
C08730=1024.545,-62.414,-92.020,166.765,47.314,158.640
C08731=1024.551,-62.164,-92.032,166.767,47.311,158.639
C08732=1024.556,-61.914,-92.043,166.770,47.308,158.639
C08733=1024.563,-61.665,-92.055,166.774,47.305,158.639
C08734=1024.569,-61.415,-92.066,166.777,47.302,158.639
C08735=1024.574,-61.166,-92.077,166.779,47.299,158.639
C08736=1024.581,-60.915,-92.088,166.782,47.296,158.639
C08737=1024.586,-60.666,-92.100,166.786,47.293,158.639
C08738=1024.592,-60.417,-92.111,166.789,47.290,158.638
C08739=1024.598,-60.167,-92.122,166.791,47.287,158.638
C08740=1024.604,-59.917,-92.133,166.794,47.284,158.638
C08741=1024.611,-59.668,-92.145,166.798,47.281,158.638
C08742=1024.616,-59.418,-92.156,166.801,47.277,158.638
C08743=1024.622,-59.168,-92.168,166.803,47.275,158.638
C08744=1024.628,-58.919,-92.180,166.806,47.271,158.637
C08745=1024.634,-58.669,-92.190,166.809,47.268,158.637
C08746=1024.640,-58.419,-92.202,166.811,47.265,158.637
C08747=1024.646,-58.169,-92.213,166.815,47.262,158.637
C08748=1024.652,-57.920,-92.225,166.818,47.259,158.637
C08749=1024.657,-57.670,-92.236,166.821,47.256,158.636
C08750=1024.664,-57.420,-92.247,166.823,47.253,158.636
C08751=1024.670,-57.171,-92.259,166.827,47.250,158.636
C08752=1024.676,-56.921,-92.270,166.830,47.246,158.636
C08753=1024.682,-56.672,-92.282,166.833,47.243,158.636
C08754=1024.688,-56.421,-92.293,166.835,47.240,158.636
C08755=1024.694,-56.172,-92.304,166.838,47.237,158.635
C08756=1024.700,-55.922,-92.316,166.841,47.234,158.635
C08757=1024.706,-55.673,-92.327,166.845,47.230,158.635
C08758=1024.712,-55.423,-92.338,166.847,47.228,158.635
C08759=1024.718,-55.174,-92.350,166.850,47.225,158.635
C08760=1024.724,-54.923,-92.362,166.853,47.221,158.634
C08761=1024.730,-54.674,-92.373,166.857,47.218,158.634
C08762=1024.736,-54.424,-92.385,166.859,47.215,158.634
C08763=1024.742,-54.175,-92.396,166.862,47.212,158.634
C08764=1024.749,-53.925,-92.408,166.865,47.209,158.634
C08765=1024.755,-53.675,-92.420,166.868,47.205,158.634
C08766=1024.760,-53.426,-92.431,166.870,47.203,158.633
C08767=1024.767,-53.146,-92.444,166.874,47.199,158.633
C08768=1024.774,-52.865,-92.457,166.878,47.195,158.633
C08769=1024.781,-52.585,-92.470,166.881,47.192,158.633
C08770=1024.788,-52.305,-92.482,166.884,47.189,158.633
C08771=1024.794,-52.055,-92.495,166.887,47.185,158.632
C08772=1024.800,-51.806,-92.506,166.890,47.182,158.632
C08773=1024.806,-51.556,-92.518,166.892,47.179,158.632
C08774=1024.812,-51.307,-92.529,166.895,47.176,158.632
C08775=1024.819,-51.057,-92.541,166.899,47.173,158.632
C08776=1024.825,-50.807,-92.553,166.901,47.170,158.631
C08777=1024.830,-50.558,-92.564,166.904,47.167,158.631
C08778=1024.836,-50.308,-92.577,166.907,47.164,158.631
C08779=1024.843,-50.058,-92.588,166.909,47.161,158.631
C08780=1024.848,-49.809,-92.600,166.913,47.158,158.631
C08781=1024.854,-49.559,-92.613,166.916,47.155,158.631
C08782=1024.860,-49.310,-92.624,166.918,47.152,158.630
C08783=1024.866,-49.026,-92.638,166.921,47.149,158.630
C08784=1024.873,-48.743,-92.651,166.925,47.145,158.630
C08785=1024.880,-48.460,-92.665,166.929,47.142,158.630
C08786=1024.887,-48.176,-92.678,166.932,47.138,158.630
C08787=1024.892,-47.927,-92.691,166.934,47.135,158.629
C08788=1024.898,-47.677,-92.703,166.938,47.133,158.629
C08789=1024.905,-47.428,-92.715,166.941,47.130,158.629
C08790=1024.910,-47.178,-92.727,166.943,47.127,158.629
C08791=1024.917,-46.928,-92.739,166.946,47.124,158.629
C08792=1024.922,-46.679,-92.751,166.949,47.121,158.629
C08793=1024.928,-46.429,-92.763,166.952,47.118,158.629
C08794=1024.934,-46.180,-92.775,166.955,47.115,158.628
C08795=1024.940,-45.930,-92.788,166.957,47.112,158.628
C08796=1024.946,-45.680,-92.799,166.960,47.109,158.628
C08797=1024.952,-45.430,-92.811,166.964,47.106,158.628
C08798=1024.958,-45.181,-92.824,166.966,47.103,158.628
C08799=1024.964,-44.932,-92.835,166.969,47.100,158.627
C08800=1024.970,-44.682,-92.848,166.971,47.097,158.627
C08801=1024.976,-44.432,-92.860,166.975,47.094,158.627
C08802=1024.982,-44.183,-92.872,166.978,47.091,158.627
C08803=1024.988,-43.933,-92.885,166.980,47.088,158.627
C08804=1024.994,-43.684,-92.897,166.983,47.085,158.627
C08805=1025.000,-43.433,-92.908,166.987,47.082,158.626
C08806=1025.005,-43.184,-92.921,166.989,47.079,158.626
C08807=1025.012,-42.934,-92.933,166.992,47.076,158.626
C08808=1025.018,-42.684,-92.945,166.994,47.073,158.626
C08809=1025.024,-42.435,-92.957,166.997,47.070,158.626
C08810=1025.030,-42.186,-92.969,167.001,47.067,158.626
C08811=1025.036,-41.936,-92.982,167.003,47.064,158.625
C08812=1025.042,-41.686,-92.994,167.006,47.061,158.625
C08813=1025.048,-41.436,-93.006,167.009,47.058,158.625
C08814=1025.054,-41.186,-93.019,167.012,47.055,158.625
C08815=1025.060,-40.938,-93.030,167.015,47.052,158.625
C08816=1025.066,-40.688,-93.043,167.018,47.049,158.624
C08817=1025.073,-40.438,-93.055,167.020,47.046,158.624
C08818=1025.079,-40.188,-93.068,167.024,47.043,158.624
C08819=1025.085,-39.938,-93.080,167.026,47.040,158.624
C08820=1025.091,-39.689,-93.092,167.029,47.037,158.624
C08821=1025.097,-39.440,-93.104,167.032,47.034,158.624
C08822=1025.102,-39.190,-93.117,167.034,47.031,158.623
C08823=1025.109,-38.940,-93.129,167.038,47.028,158.623
C08824=1025.115,-38.691,-93.142,167.040,47.025,158.623
C08825=1025.121,-38.441,-93.155,167.043,47.022,158.623
C08826=1025.127,-38.192,-93.167,167.047,47.020,158.623
C08827=1025.132,-37.943,-93.180,167.049,47.017,158.623
C08828=1025.138,-37.695,-93.192,167.052,47.014,158.622
C08829=1025.144,-37.448,-93.204,167.054,47.011,158.622
C08830=1025.150,-37.200,-93.218,167.058,47.008,158.622
C08831=1025.156,-36.952,-93.229,167.060,47.005,158.622
C08832=1025.162,-36.704,-93.242,167.063,47.002,158.622
C08833=1025.167,-36.456,-93.254,167.066,47.000,158.622
C08834=1025.174,-36.208,-93.267,167.069,46.997,158.621
C08835=1025.180,-35.959,-93.280,167.071,46.994,158.621
C08836=1025.186,-35.709,-93.292,167.074,46.991,158.621
C08837=1025.192,-35.459,-93.305,167.076,46.988,158.621
C08838=1025.199,-35.210,-93.318,167.080,46.985,158.621
C08839=1025.204,-34.961,-93.330,167.083,46.982,158.621
C08840=1025.210,-34.711,-93.342,167.085,46.979,158.620
C08841=1025.216,-34.461,-93.355,167.088,46.976,158.620
C08842=1025.222,-34.212,-93.368,167.091,46.973,158.620
C08843=1025.228,-33.962,-93.381,167.094,46.971,158.620
C08844=1025.234,-33.712,-93.393,167.096,46.968,158.620
C08845=1025.240,-33.463,-93.407,167.100,46.965,158.620
C08846=1025.246,-33.213,-93.419,167.102,46.962,158.619
C08847=1025.252,-32.963,-93.432,167.105,46.959,158.619
C08848=1025.258,-32.714,-93.445,167.108,46.956,158.619
C08849=1025.265,-32.464,-93.457,167.111,46.953,158.619
C08850=1025.271,-32.214,-93.470,167.114,46.950,158.619
C08851=1025.277,-31.965,-93.483,167.116,46.947,158.618
C08852=1025.282,-31.716,-93.495,167.119,46.944,158.618
C08853=1025.288,-31.466,-93.508,167.121,46.942,158.618
C08854=1025.294,-31.216,-93.521,167.125,46.938,158.618
C08855=1025.300,-30.967,-93.533,167.128,46.935,158.618
C08856=1025.306,-30.717,-93.547,167.130,46.933,158.617
C08857=1025.312,-30.467,-93.559,167.133,46.929,158.617
C08858=1025.318,-30.218,-93.572,167.136,46.927,158.617
C08859=1025.324,-29.968,-93.585,167.139,46.924,158.617
C08860=1025.330,-29.718,-93.598,167.141,46.921,158.617
C08861=1025.336,-29.469,-93.611,167.144,46.918,158.617
C08862=1025.342,-29.219,-93.623,167.147,46.915,158.616
C08863=1025.349,-28.970,-93.636,167.150,46.912,158.616
C08864=1025.355,-28.720,-93.649,167.153,46.909,158.616
C08865=1025.361,-28.471,-93.662,167.155,46.906,158.616
C08866=1025.368,-28.221,-93.675,167.159,46.903,158.616
C08867=1025.374,-27.971,-93.688,167.161,46.900,158.615
C08868=1025.380,-27.721,-93.701,167.164,46.897,158.615
C08869=1025.386,-27.472,-93.714,167.166,46.894,158.615
C08870=1025.392,-27.222,-93.726,167.169,46.891,158.615
C08871=1025.398,-26.973,-93.740,167.172,46.889,158.615
C08872=1025.404,-26.723,-93.753,167.175,46.886,158.615
C08873=1025.410,-26.474,-93.766,167.177,46.883,158.614
C08874=1025.416,-26.224,-93.779,167.181,46.880,158.614
C08875=1025.422,-25.974,-93.792,167.183,46.877,158.614
C08876=1025.428,-25.725,-93.805,167.186,46.874,158.614
C08877=1025.434,-25.476,-93.819,167.188,46.871,158.614
C08878=1025.440,-25.226,-93.832,167.192,46.869,158.614
C08879=1025.446,-24.976,-93.845,167.194,46.866,158.613
C08880=1025.452,-24.727,-93.858,167.197,46.863,158.613
C08881=1025.458,-24.477,-93.871,167.200,46.860,158.613
C08882=1025.463,-24.228,-93.885,167.203,46.857,158.613
C08883=1025.470,-23.978,-93.898,167.205,46.854,158.613
C08884=1025.476,-23.728,-93.911,167.208,46.851,158.612
C08885=1025.482,-23.479,-93.924,167.211,46.849,158.612
C08886=1025.488,-23.229,-93.938,167.214,46.846,158.612
C08887=1025.494,-22.980,-93.951,167.216,46.843,158.612
C08888=1025.500,-22.730,-93.964,167.220,46.840,158.612
C08889=1025.506,-22.481,-93.977,167.222,46.837,158.611
C08890=1025.512,-22.231,-93.990,167.225,46.834,158.611
C08891=1025.518,-21.982,-94.004,167.227,46.832,158.611
C08892=1025.524,-21.731,-94.017,167.230,46.828,158.611
C08893=1025.531,-21.482,-94.030,167.233,46.826,158.611
C08894=1025.537,-21.233,-94.044,167.236,46.823,158.611
C08895=1025.543,-20.952,-94.059,167.238,46.820,158.610
C08896=1025.550,-20.672,-94.073,167.241,46.817,158.610
C08897=1025.557,-20.390,-94.089,167.245,46.814,158.610
C08898=1025.564,-20.110,-94.104,167.248,46.810,158.610
C08899=1025.570,-19.861,-94.117,167.251,46.807,158.610
C08900=1025.575,-19.611,-94.130,167.253,46.804,158.609
C08901=1025.582,-19.361,-94.144,167.256,46.801,158.609
C08902=1025.588,-19.112,-94.157,167.259,46.798,158.609
C08903=1025.594,-18.862,-94.170,167.262,46.796,158.609
C08904=1025.600,-18.613,-94.184,167.264,46.793,158.609
C08905=1025.606,-18.364,-94.197,167.268,46.790,158.608
C08906=1025.613,-18.114,-94.211,167.270,46.787,158.608
C08907=1025.619,-17.864,-94.224,167.273,46.784,158.608
C08908=1025.625,-17.614,-94.237,167.275,46.781,158.608
C08909=1025.631,-17.365,-94.251,167.279,46.778,158.608
C08910=1025.637,-17.115,-94.264,167.281,46.775,158.607
C08911=1025.644,-16.866,-94.277,167.284,46.772,158.607
C08912=1025.650,-16.616,-94.291,167.286,46.770,158.607
C08913=1025.655,-16.367,-94.305,167.289,46.766,158.607
C08914=1025.662,-16.117,-94.318,167.292,46.764,158.607
C08915=1025.668,-15.868,-94.332,167.295,46.761,158.606
C08916=1025.674,-15.618,-94.345,167.297,46.758,158.606
C08917=1025.680,-15.369,-94.359,167.299,46.755,158.606
C08918=1025.686,-15.118,-94.373,167.303,46.752,158.606
C08919=1025.692,-14.869,-94.386,167.305,46.749,158.606
C08920=1025.698,-14.620,-94.400,167.308,46.747,158.606
C08921=1025.704,-14.370,-94.413,167.311,46.744,158.605
C08922=1025.710,-14.120,-94.428,167.313,46.741,158.605
C08923=1025.716,-13.871,-94.441,167.316,46.738,158.605
C08924=1025.722,-13.621,-94.455,167.318,46.735,158.605
C08925=1025.729,-13.371,-94.468,167.322,46.732,158.605
C08926=1025.734,-13.122,-94.483,167.324,46.730,158.604
C08927=1025.741,-12.873,-94.496,167.327,46.727,158.604
C08928=1025.746,-12.624,-94.510,167.330,46.724,158.604
C08929=1025.753,-12.374,-94.524,167.332,46.722,158.604
C08930=1025.758,-12.124,-94.538,167.335,46.718,158.604
C08931=1025.765,-11.875,-94.551,167.337,46.716,158.603
C08932=1025.771,-11.624,-94.565,167.341,46.713,158.603
C08933=1025.777,-11.376,-94.579,167.343,46.710,158.603
C08934=1025.783,-11.126,-94.593,167.345,46.708,158.603
C08935=1025.789,-10.876,-94.607,167.349,46.705,158.603
C08936=1025.795,-10.627,-94.620,167.351,46.702,158.602
C08937=1025.801,-10.377,-94.634,167.354,46.699,158.602
C08938=1025.807,-10.128,-94.649,167.356,46.696,158.602
C08939=1025.814,-9.878,-94.662,167.360,46.693,158.602
C08940=1025.819,-9.629,-94.676,167.362,46.690,158.602
C08941=1025.826,-9.379,-94.689,167.364,46.687,158.601
C08942=1025.831,-9.129,-94.703,167.367,46.684,158.601
C08943=1025.837,-8.880,-94.718,167.369,46.682,158.601
C08944=1025.844,-8.630,-94.731,167.373,46.679,158.601
C08945=1025.850,-8.381,-94.745,167.375,46.676,158.601
C08946=1025.856,-8.131,-94.759,167.378,46.673,158.601
C08947=1025.862,-7.882,-94.774,167.381,46.671,158.600
///RCONF 1,0,0,0,0,0,0,0,0,0,0,0,0,0,0,0,0,0,0,0,0,0,0,0
C08948=1025.868,-7.633,-94.787,167.383,46.668,158.600
C08949=1025.874,-7.382,-94.801,167.386,46.665,158.600
C08950=1025.881,-7.134,-94.815,167.388,46.662,158.600
C08951=1025.887,-6.883,-94.829,167.392,46.659,158.600
C08952=1025.893,-6.634,-94.842,167.394,46.656,158.599
C08953=1025.899,-6.385,-94.856,167.396,46.653,158.599
C08954=1025.906,-6.135,-94.871,167.399,46.650,158.599
C08955=1025.911,-5.886,-94.885,167.402,46.647,158.599
C08956=1025.917,-5.635,-94.899,167.405,46.644,158.598
C08957=1025.924,-5.387,-94.913,167.407,46.642,158.598
C08958=1025.930,-5.137,-94.927,167.410,46.639,158.598
C08959=1025.937,-4.855,-94.942,167.413,46.636,158.598
C08960=1025.944,-4.573,-94.958,167.416,46.633,158.598
C08961=1025.951,-4.290,-94.974,167.419,46.629,158.597
C08962=1025.958,-4.008,-94.990,167.422,46.626,158.597
C08963=1025.964,-3.758,-95.004,167.424,46.623,158.597
C08964=1025.970,-3.509,-95.019,167.428,46.620,158.597
C08965=1025.976,-3.259,-95.033,167.430,46.618,158.597
C08966=1025.982,-3.010,-95.048,167.432,46.615,158.596
C08967=1025.988,-2.760,-95.062,167.436,46.612,158.596
C08968=1025.994,-2.511,-95.077,167.438,46.609,158.596
C08969=1026.001,-2.261,-95.090,167.440,46.607,158.596
C08970=1026.006,-2.012,-95.105,167.444,46.604,158.596
C08971=1026.012,-1.762,-95.119,167.446,46.601,158.596
C08972=1026.018,-1.513,-95.134,167.448,46.599,158.595
C08973=1026.024,-1.264,-95.148,167.451,46.596,158.595
C08974=1026.030,-1.013,-95.163,167.454,46.593,158.595
C08975=1026.036,-0.764,-95.177,167.456,46.591,158.595
C08976=1026.042,-0.514,-95.191,167.459,46.588,158.595
C08977=1026.048,-0.265,-95.206,167.462,46.585,158.594
C08978=1026.055,-0.016,-95.220,167.464,46.582,158.594
C08979=1026.060,0.234,-95.234,167.467,46.579,158.594
C08980=1026.067,0.483,-95.249,167.470,46.577,158.594
C08981=1026.072,0.733,-95.263,167.472,46.574,158.594
C08982=1026.079,0.983,-95.278,167.475,46.571,158.593
C08983=1026.084,1.232,-95.292,167.477,46.568,158.593
C08984=1026.090,1.482,-95.307,167.479,46.566,158.593
C08985=1026.096,1.731,-95.321,167.483,46.563,158.593
C08986=1026.103,1.981,-95.336,167.485,46.560,158.593
